METHOD INTERNAL ParseResponsePayload : DINT
VAR_INPUT
  /// Response data
  ResponseData : RobotLibraryRecvDataFB;
  /// Timestamp
  Timestamp    : SystemTime;  
END_VAR
// Table 6-566: Received CMD payload (RC to PLC) of "MeasuringInput"
// --------------------------
// Header
// --------------------------
// Byte 000 : USINT - ParSeq | State     
// Byte 001 : SINT  - AlarmMessageSeverity    
// Byte 002 : UINT  - AlarmMessageCode HB
// Byte 003 :       - AlarmMessageCode LB
// --------------------------
// Datablock
// --------------------------
// Byte 004 : BOOL      - Enabled
// Byte 005 : UINT      - MeasuringID LW LB 
// Byte 006 : USINT     - ToolNo_1
// Byte 007 : USINT     - FrameNo_1
// Byte 008 : USINT     - ToolNo_2
// Byte 009 : USINT     - FrameNo_2
// Byte 010 : REAL      - MeasuredCartesianPosition_1.X HW HB
// Byte 011 :           - MeasuredCartesianPosition_1.X HW LB
// Byte 012 :           - MeasuredCartesianPosition_1.X LW HB
// Byte 013 :           - MeasuredCartesianPosition_1.X LW LB
// Byte 014 : REAL      - MeasuredCartesianPosition_1.Y HW HB
// Byte 015 :           - MeasuredCartesianPosition_1.Y HW LB
// Byte 016 :           - MeasuredCartesianPosition_1.Y LW HB
// Byte 017 :           - MeasuredCartesianPosition_1.Y LW LB
// Byte 018 : REAL      - MeasuredCartesianPosition_1.Z HW HB
// Byte 019 :           - MeasuredCartesianPosition_1.Z HW LB
// Byte 020 :           - MeasuredCartesianPosition_1.Z LW HB
// Byte 021 :           - MeasuredCartesianPosition_1.Z LW LB
// Byte 022 : REAL      - MeasuredCartesianPosition_1.Rx HW HB
// Byte 023 :           - MeasuredCartesianPosition_1.Rx HW LB
// Byte 024 :           - MeasuredCartesianPosition_1.Rx LW HB
// Byte 025 :           - MeasuredCartesianPosition_1.Rx LW LB
// Byte 026 : REAL      - MeasuredCartesianPosition_1.Ry HW HB
// Byte 027 :           - MeasuredCartesianPosition_1.Ry HW LB
// Byte 028 :           - MeasuredCartesianPosition_1.Ry LW HB
// Byte 029 :           - MeasuredCartesianPosition_1.Ry LW LB
// Byte 030 : REAL      - MeasuredCartesianPosition_1.Rz HW HB
// Byte 031 :           - MeasuredCartesianPosition_1.Rz HW LB
// Byte 032 :           - MeasuredCartesianPosition_1.Rz LW HB
// Byte 033 :           - MeasuredCartesianPosition_1.Rz LW LB
// Byte 034 : Config    - MeasuredCartesianPosition_1.ArmConfig
// Byte 035 :           - MeasuredCartesianPosition_1.Reserve
// Byte 036 : TurnNumber- MeasuredCartesianPosition_1.TurnNumber.J1 + J2  HW HB
// Byte 037 :           - MeasuredCartesianPosition_1.TurnNumber.J3 + J4  HW LB
// Byte 038 :           - MeasuredCartesianPosition_1.TurnNumber.J5 + J6  LW LB
// Byte 039 :           - MeasuredCartesianPosition_1.TurnNumber.E1       LW LB
// Byte 040 : REAL      - MeasuredCartesianPosition_1.E1 HW HB
// Byte 041 :           - MeasuredCartesianPosition_1.E1 HW LB
// Byte 042 :           - MeasuredCartesianPosition_1.E1 LW HB
// Byte 043 :           - MeasuredCartesianPosition_1.E1 LW LB
// Byte 044 : REAL      - MeasuredJointPosition_1.J1 HW HB
// Byte 045 :           - MeasuredJointPosition_1.J1 HW LB
// Byte 046 :           - MeasuredJointPosition_1.J1 LW HB
// Byte 047 :           - MeasuredJointPosition_1.J1 LW LB
// Byte 048 : REAL      - MeasuredJointPosition_1.J2 HW HB
// Byte 049 :           - MeasuredJointPosition_1.J2 HW LB
// Byte 050 :           - MeasuredJointPosition_1.J2 LW HB
// Byte 051 :           - MeasuredJointPosition_1.J2 LW LB
// Byte 052 : REAL      - MeasuredJointPosition_1.J3 HW HB
// Byte 053 :           - MeasuredJointPosition_1.J3 HW LB
// Byte 054 :           - MeasuredJointPosition_1.J3 LW HB
// Byte 055 :           - MeasuredJointPosition_1.J3 LW LB
// Byte 056 : REAL      - MeasuredJointPosition_1.J4 HW HB
// Byte 057 :           - MeasuredJointPosition_1.J4 HW LB
// Byte 058 :           - MeasuredJointPosition_1.J4 LW HB
// Byte 059 :           - MeasuredJointPosition_1.J4 LW LB
// Byte 060 : REAL      - MeasuredJointPosition_1.J5 HW HB
// Byte 061 :           - MeasuredJointPosition_1.J5 HW LB
// Byte 062 :           - MeasuredJointPosition_1.J5 LW HB
// Byte 063 :           - MeasuredJointPosition_1.J5 LW LB
// Byte 064 : REAL      - MeasuredJointPosition_1.J6 HW HB
// Byte 065 :           - MeasuredJointPosition_1.J6 HW LB
// Byte 066 :           - MeasuredJointPosition_1.J6 LW HB
// Byte 067 :           - MeasuredJointPosition_1.J6 LW LB
// Byte 068 : REAL      - MeasuredJointPosition_1.E1 HW HB
// Byte 069 :           - MeasuredJointPosition_1.E1 HW LB
// Byte 070 :           - MeasuredJointPosition_1.E1 LW HB
// Byte 071 :           - MeasuredJointPosition_1.E1 LW LB
// Byte 072 : REAL      - MeasuredCartesianPosition_2.X HW HB
// Byte 073 :           - MeasuredCartesianPosition_2.X HW LB
// Byte 074 :           - MeasuredCartesianPosition_2.X LW HB
// Byte 075 :           - MeasuredCartesianPosition_2.X LW LB
// Byte 076 : REAL      - MeasuredCartesianPosition_2.Y HW HB
// Byte 077 :           - MeasuredCartesianPosition_2.Y HW LB
// Byte 078 :           - MeasuredCartesianPosition_2.Y LW HB
// Byte 079 :           - MeasuredCartesianPosition_2.Y LW LB
// Byte 080 : REAL      - MeasuredCartesianPosition_2.Z HW HB
// Byte 081 :           - MeasuredCartesianPosition_2.Z HW LB
// Byte 082 :           - MeasuredCartesianPosition_2.Z LW HB
// Byte 083 :           - MeasuredCartesianPosition_2.Z LW LB
// Byte 084 : REAL      - MeasuredCartesianPosition_2.Rx HW HB
// Byte 085 :           - MeasuredCartesianPosition_2.Rx HW LB
// Byte 086 :           - MeasuredCartesianPosition_2.Rx LW HB
// Byte 087 :           - MeasuredCartesianPosition_2.Rx LW LB
// Byte 088 : REAL      - MeasuredCartesianPosition_2.Ry HW HB
// Byte 089 :           - MeasuredCartesianPosition_2.Ry HW LB
// Byte 090 :           - MeasuredCartesianPosition_2.Ry LW HB
// Byte 091 :           - MeasuredCartesianPosition_2.Ry LW LB
// Byte 092 : REAL      - MeasuredCartesianPosition_2.Rz HW HB
// Byte 093 :           - MeasuredCartesianPosition_2.Rz HW LB
// Byte 094 :           - MeasuredCartesianPosition_2.Rz LW HB
// Byte 095 :           - MeasuredCartesianPosition_2.Rz LW LB
// Byte 096 : Config    - MeasuredCartesianPosition_2.ArmConfig
// Byte 097 :           - MeasuredCartesianPosition_2.Reserve
// Byte 098 : TurnNumber- MeasuredCartesianPosition_2.TurnNumber.J1 + J2  HW HB
// Byte 099 :           - MeasuredCartesianPosition_2.TurnNumber.J3 + J4  HW LB
// Byte 100 :           - MeasuredCartesianPosition_2.TurnNumber.J5 + J6  LW LB
// Byte 101 :           - MeasuredCartesianPosition_2.TurnNumber.E1       LW LB
// Byte 102 : REAL      - MeasuredCartesianPosition_2.E1 HW HB
// Byte 103 :           - MeasuredCartesianPosition_2.E1 HW LB
// Byte 104 :           - MeasuredCartesianPosition_2.E1 LW HB
// Byte 105 :           - MeasuredCartesianPosition_2.E1 LW LB
// Byte 106 : REAL      - MeasuredJointPosition_2.J1 HW HB
// Byte 107 :           - MeasuredJointPosition_2.J1 HW LB
// Byte 108 :           - MeasuredJointPosition_2.J1 LW HB
// Byte 109 :           - MeasuredJointPosition_2.J1 LW LB
// Byte 110 : REAL      - MeasuredJointPosition_2.J2 HW HB
// Byte 111 :           - MeasuredJointPosition_2.J2 HW LB
// Byte 112 :           - MeasuredJointPosition_2.J2 LW HB
// Byte 113 :           - MeasuredJointPosition_2.J2 LW LB
// Byte 114 : REAL      - MeasuredJointPosition_2.J3 HW HB
// Byte 115 :           - MeasuredJointPosition_2.J3 HW LB
// Byte 116 :           - MeasuredJointPosition_2.J3 LW HB
// Byte 117 :           - MeasuredJointPosition_2.J3 LW LB
// Byte 118 : REAL      - MeasuredJointPosition_2.J4 HW HB
// Byte 119 :           - MeasuredJointPosition_2.J4 HW LB
// Byte 120 :           - MeasuredJointPosition_2.J4 LW HB
// Byte 121 :           - MeasuredJointPosition_2.J4 LW LB
// Byte 122 : REAL      - MeasuredJointPosition_2.J5 HW HB
// Byte 123 :           - MeasuredJointPosition_2.J5 HW LB
// Byte 124 :           - MeasuredJointPosition_2.J5 LW HB
// Byte 125 :           - MeasuredJointPosition_2.J5 LW LB
// Byte 126 : REAL      - MeasuredJointPosition_2.J6 HW HB
// Byte 127 :           - MeasuredJointPosition_2.J6 HW LB
// Byte 128 :           - MeasuredJointPosition_2.J6 LW HB
// Byte 129 :           - MeasuredJointPosition_2.J6 LW LB
// Byte 130 : REAL      - MeasuredJointPosition_2.E1 HW HB
// Byte 131 :           - MeasuredJointPosition_2.E1 HW LB
// Byte 132 :           - MeasuredJointPosition_2.E1 LW HB
// Byte 133 :           - MeasuredJointPosition_2.E1 LW LB
// Byte 134 : REAL      - MeasuredCartesianPosition_1.E2 HW HB
// Byte 135 :           - MeasuredCartesianPosition_1.E2 HW LB
// Byte 136 :           - MeasuredCartesianPosition_1.E2 LW HB
// Byte 137 :           - MeasuredCartesianPosition_1.E2 LW LB
// Byte 138 : REAL      - MeasuredCartesianPosition_1.E3 HW HB
// Byte 139 :           - MeasuredCartesianPosition_1.E3 HW LB
// Byte 140 :           - MeasuredCartesianPosition_1.E3 LW HB
// Byte 141 :           - MeasuredCartesianPosition_1.E3 LW LB
// Byte 142 : REAL      - MeasuredCartesianPosition_1.E4 HW HB
// Byte 143 :           - MeasuredCartesianPosition_1.E4 HW LB
// Byte 144 :           - MeasuredCartesianPosition_1.E4 LW HB
// Byte 145 :           - MeasuredCartesianPosition_1.E4 LW LB
// Byte 146 : REAL      - MeasuredCartesianPosition_1.E5 HW HB
// Byte 147 :           - MeasuredCartesianPosition_1.E5 HW LB
// Byte 148 :           - MeasuredCartesianPosition_1.E5 LW HB
// Byte 149 :           - MeasuredCartesianPosition_1.E5 LW LB
// Byte 150 : REAL      - MeasuredCartesianPosition_1.E6 HW HB
// Byte 151 :           - MeasuredCartesianPosition_1.E6 HW LB
// Byte 152 :           - MeasuredCartesianPosition_1.E6 LW HB
// Byte 153 :           - MeasuredCartesianPosition_1.E6 LW LB
// Byte 154 : REAL      - MeasuredJointPosition_1.E2 HW HB
// Byte 155 :           - MeasuredJointPosition_1.E2 HW LB
// Byte 156 :           - MeasuredJointPosition_1.E2 LW HB
// Byte 157 :           - MeasuredJointPosition_1.E2 LW LB
// Byte 158 : REAL      - MeasuredJointPosition_1.E3 HW HB
// Byte 159 :           - MeasuredJointPosition_1.E3 HW LB
// Byte 160 :           - MeasuredJointPosition_1.E3 LW HB
// Byte 161 :           - MeasuredJointPosition_1.E3 LW LB
// Byte 162 : REAL      - MeasuredJointPosition_1.E4 HW HB
// Byte 163 :           - MeasuredJointPosition_1.E4 HW LB
// Byte 164 :           - MeasuredJointPosition_1.E4 LW HB
// Byte 165 :           - MeasuredJointPosition_1.E4 LW LB
// Byte 166 : REAL      - MeasuredJointPosition_1.E5 HW HB
// Byte 167 :           - MeasuredJointPosition_1.E5 HW LB
// Byte 168 :           - MeasuredJointPosition_1.E5 LW HB
// Byte 169 :           - MeasuredJointPosition_1.E5 LW LB
// Byte 170 : REAL      - MeasuredJointPosition_1.E6 HW HB
// Byte 171 :           - MeasuredJointPosition_1.E6 HW LB
// Byte 172 :           - MeasuredJointPosition_1.E6 LW HB
// Byte 173 :           - MeasuredJointPosition_1.E6 LW LB
// Byte 174 : REAL      - MeasuredCartesianPosition_2.E2 HW HB
// Byte 175 :           - MeasuredCartesianPosition_2.E2 HW LB
// Byte 176 :           - MeasuredCartesianPosition_2.E2 LW HB
// Byte 177 :           - MeasuredCartesianPosition_2.E2 LW LB
// Byte 178 : REAL      - MeasuredCartesianPosition_2.E3 HW HB
// Byte 179 :           - MeasuredCartesianPosition_2.E3 HW LB
// Byte 180 :           - MeasuredCartesianPosition_2.E3 LW HB
// Byte 181 :           - MeasuredCartesianPosition_2.E3 LW LB
// Byte 182 : REAL      - MeasuredCartesianPosition_2.E4 HW HB
// Byte 183 :           - MeasuredCartesianPosition_2.E4 HW LB
// Byte 184 :           - MeasuredCartesianPosition_2.E4 LW HB
// Byte 185 :           - MeasuredCartesianPosition_2.E4 LW LB
// Byte 186 : REAL      - MeasuredCartesianPosition_2.E5 HW HB
// Byte 187 :           - MeasuredCartesianPosition_2.E5 HW LB
// Byte 188 :           - MeasuredCartesianPosition_2.E5 LW HB
// Byte 189 :           - MeasuredCartesianPosition_2.E5 LW LB
// Byte 190 : REAL      - MeasuredCartesianPosition_2.E6 HW HB
// Byte 191 :           - MeasuredCartesianPosition_2.E6 HW LB
// Byte 192 :           - MeasuredCartesianPosition_2.E6 LW HB
// Byte 193 :           - MeasuredCartesianPosition_2.E6 LW LB
// Byte 194 : REAL      - MeasuredJointPosition_2.E2 HW HB
// Byte 195 :           - MeasuredJointPosition_2.E2 HW LB
// Byte 196 :           - MeasuredJointPosition_2.E2 LW HB
// Byte 197 :           - MeasuredJointPosition_2.E2 LW LB
// Byte 198 : REAL      - MeasuredJointPosition_2.E3 HW HB
// Byte 199 :           - MeasuredJointPosition_2.E3 HW LB
// Byte 200 :           - MeasuredJointPosition_2.E3 LW HB
// Byte 201 :           - MeasuredJointPosition_2.E3 LW LB
// Byte 202 : REAL      - MeasuredJointPosition_2.E4 HW HB
// Byte 203 :           - MeasuredJointPosition_2.E4 HW LB
// Byte 204 :           - MeasuredJointPosition_2.E4 LW HB
// Byte 205 :           - MeasuredJointPosition_2.E4 LW LB
// Byte 206 : REAL      - MeasuredJointPosition_2.E5 HW HB
// Byte 207 :           - MeasuredJointPosition_2.E5 HW LB
// Byte 208 :           - MeasuredJointPosition_2.E5 LW HB
// Byte 209 :           - MeasuredJointPosition_2.E5 LW LB
// Byte 210 : REAL      - MeasuredJointPosition_2.E6 HW HB
// Byte 211 :           - MeasuredJointPosition_2.E6 HW LB
// Byte 212 :           - MeasuredJointPosition_2.E6 LW HB
// Byte 213 :           - MeasuredJointPosition_2.E6 LW LB
// call base implementation to parse the header from payload buffer
ResponseData.PayloadPtr := SUPER^.ParseResponsePayload(ResponseData := ResponseData, Timestamp := Timestamp);

// copy parsed header to response
_response.ParSeq               := _rspHeader.ParSeq;
_response.State                := _rspHeader.State;
_response.AlarmMessageSeverity := _rspHeader.AlarmMessageSeverity;
_response.AlarmMessageCode     := _rspHeader.AlarmMessageCode;


// Get Response.MeasuringID
_response.MeasuringID   := ResponseData.GetUint();
// Get Response.Measurings[1].ToolNo
_response.Measurings[1].ToolNo := ResponseData.GetUsint();
// Get Response.Measurings[1].FrameNo
_response.Measurings[1].FrameNo := ResponseData.GetUsint();
// Get Response.Measurings[2].ToolNo
_response.Measurings[2].ToolNo := ResponseData.GetUsint();
// Get Response.Measurings[2].FrameNo
_response.Measurings[2].FrameNo := ResponseData.GetUsint();
// Get Response.Measurings[1].MeasuredCartesianPosition.X
_response.Measurings[1].MeasuredCartesianPosition.X := ResponseData.GetReal();
// Get Response.Measurings[1].MeasuredCartesianPosition.Y
_response.Measurings[1].MeasuredCartesianPosition.Y := ResponseData.GetReal();
// Get Response.Measurings[1].MeasuredCartesianPosition.Z
_response.Measurings[1].MeasuredCartesianPosition.Z := ResponseData.GetReal();
// Get Response.Measurings[1].MeasuredCartesianPosition.Rx
_response.Measurings[1].MeasuredCartesianPosition.Rx := ResponseData.GetReal();
// Get Response.Measurings[1].MeasuredCartesianPosition.Ry
_response.Measurings[1].MeasuredCartesianPosition.Ry := ResponseData.GetReal();
// Get Response.Measurings[1].MeasuredCartesianPosition.Rz
_response.Measurings[1].MeasuredCartesianPosition.Rz := ResponseData.GetReal();
// Get Response.Measurings[1].MeasuredCartesianPosition.Config
_response.Measurings[1].MeasuredCartesianPosition.Config := ResponseData.GetArmConfig();
// Get Response.Measurings[1].MeasuredCartesianPosition.TurnNumber
_response.Measurings[1].MeasuredCartesianPosition.TurnNumber := ResponseData.GetTurnNumbers();
// Get Response.Measurings[1].MeasuredCartesianPosition.E1
_response.Measurings[1].MeasuredCartesianPosition.E1 := ResponseData.GetReal();
// Get Response.Measurings[1].MeasuredJointPosition.J1
_response.Measurings[1].MeasuredJointPosition.J1 := ResponseData.GetReal();
// Get Response.Measurings[1].MeasuredJointPosition.J2
_response.Measurings[1].MeasuredJointPosition.J2 := ResponseData.GetReal();
// Get Response.Measurings[1].MeasuredJointPosition.J3
_response.Measurings[1].MeasuredJointPosition.J3 := ResponseData.GetReal();
// Get Response.Measurings[1].MeasuredJointPosition.J4
_response.Measurings[1].MeasuredJointPosition.J4 := ResponseData.GetReal();
// Get Response.Measurings[1].MeasuredJointPosition.J5
_response.Measurings[1].MeasuredJointPosition.J5 := ResponseData.GetReal();
// Get Response.Measurings[1].MeasuredJointPosition.J6
_response.Measurings[1].MeasuredJointPosition.J6 := ResponseData.GetReal();
// Get Response.Measurings[1].MeasuredJointPosition.E1
_response.Measurings[1].MeasuredJointPosition.E1 := ResponseData.GetReal();
// Get Response.Measurings[2].MeasuredCartesianPosition.X
_response.Measurings[2].MeasuredCartesianPosition.X := ResponseData.GetReal();
// Get Response.Measurings[2].MeasuredCartesianPosition.Y
_response.Measurings[2].MeasuredCartesianPosition.Y := ResponseData.GetReal();
// Get Response.Measurings[2].MeasuredCartesianPosition.Z
_response.Measurings[2].MeasuredCartesianPosition.Z := ResponseData.GetReal();
// Get Response.Measurings[2].MeasuredCartesianPosition.Rx
_response.Measurings[2].MeasuredCartesianPosition.Rx := ResponseData.GetReal();
// Get Response.Measurings[2].MeasuredCartesianPosition.Ry
_response.Measurings[2].MeasuredCartesianPosition.Ry := ResponseData.GetReal();
// Get Response.Measurings[2].MeasuredCartesianPosition.Rz
_response.Measurings[2].MeasuredCartesianPosition.Rz := ResponseData.GetReal();
// Get Response.Measurings[2].MeasuredCartesianPosition.Config
_response.Measurings[2].MeasuredCartesianPosition.Config := ResponseData.GetArmConfig();
// Get Response.Measurings[2].MeasuredCartesianPosition.TurnNumber
_response.Measurings[2].MeasuredCartesianPosition.TurnNumber := ResponseData.GetTurnNumbers();
// Get Response.Measurings[2].MeasuredCartesianPosition.E1
_response.Measurings[2].MeasuredCartesianPosition.E1 := ResponseData.GetReal();
// Get Response.Measurings[2].MeasuredJointPosition.J1
_response.Measurings[2].MeasuredJointPosition.J1 := ResponseData.GetReal();
// Get Response.Measurings[2].MeasuredJointPosition.J2
_response.Measurings[2].MeasuredJointPosition.J2 := ResponseData.GetReal();
// Get Response.Measurings[2].MeasuredJointPosition.J3
_response.Measurings[2].MeasuredJointPosition.J3 := ResponseData.GetReal();
// Get Response.Measurings[2].MeasuredJointPosition.J4
_response.Measurings[2].MeasuredJointPosition.J4 := ResponseData.GetReal();
// Get Response.Measurings[2].MeasuredJointPosition.J5
_response.Measurings[2].MeasuredJointPosition.J5 := ResponseData.GetReal();
// Get Response.Measurings[2].MeasuredJointPosition.J6
_response.Measurings[2].MeasuredJointPosition.J6 := ResponseData.GetReal();
// Get Response.Measurings[2].MeasuredJointPosition.E1
_response.Measurings[2].MeasuredJointPosition.E1 := ResponseData.GetReal();
// Get Response.Measurings[1].MeasuredCartesianPosition.E2
_response.Measurings[1].MeasuredCartesianPosition.E2 := ResponseData.GetReal();
// Get Response.Measurings[1].MeasuredCartesianPosition.E3
_response.Measurings[1].MeasuredCartesianPosition.E3 := ResponseData.GetReal();
// Get Response.Measurings[1].MeasuredCartesianPosition.E4
_response.Measurings[1].MeasuredCartesianPosition.E4 := ResponseData.GetReal();
// Get Response.Measurings[1].MeasuredCartesianPosition.E5
_response.Measurings[1].MeasuredCartesianPosition.E5 := ResponseData.GetReal();
// Get Response.Measurings[1].MeasuredCartesianPosition.E6
_response.Measurings[1].MeasuredCartesianPosition.E6 := ResponseData.GetReal();
// Get Response.Measurings[1].MeasuredJointPosition.E2
_response.Measurings[1].MeasuredJointPosition.E2 := ResponseData.GetReal();
// Get Response.Measurings[1].MeasuredJointPosition.E3
_response.Measurings[1].MeasuredJointPosition.E3 := ResponseData.GetReal();
// Get Response.Measurings[1].MeasuredJointPosition.E4
_response.Measurings[1].MeasuredJointPosition.E4 := ResponseData.GetReal();
// Get Response.Measurings[1].MeasuredJointPosition.E5
_response.Measurings[1].MeasuredJointPosition.E5 := ResponseData.GetReal();
// Get Response.Measurings[1].MeasuredJointPosition.E6
_response.Measurings[1].MeasuredJointPosition.E6 := ResponseData.GetReal();
// Get Response.Measurings[2].MeasuredCartesianPosition.E2
_response.Measurings[2].MeasuredCartesianPosition.E2 := ResponseData.GetReal();
// Get Response.Measurings[2].MeasuredCartesianPosition.E3
_response.Measurings[2].MeasuredCartesianPosition.E3 := ResponseData.GetReal();
// Get Response.Measurings[2].MeasuredCartesianPosition.E4
_response.Measurings[2].MeasuredCartesianPosition.E4 := ResponseData.GetReal();
// Get Response.Measurings[2].MeasuredCartesianPosition.E5
_response.Measurings[2].MeasuredCartesianPosition.E5 := ResponseData.GetReal();
// Get Response.Measurings[2].MeasuredCartesianPosition.E6
_response.Measurings[2].MeasuredCartesianPosition.E6 := ResponseData.GetReal();
// Get Response.Measurings[2].MeasuredJointPosition.E2
_response.Measurings[2].MeasuredJointPosition.E2 := ResponseData.GetReal();
// Get Response.Measurings[2].MeasuredJointPosition.E3
_response.Measurings[2].MeasuredJointPosition.E3 := ResponseData.GetReal();
// Get Response.Measurings[2].MeasuredJointPosition.E4
_response.Measurings[2].MeasuredJointPosition.E4 := ResponseData.GetReal();
// Get Response.Measurings[2].MeasuredJointPosition.E5
_response.Measurings[2].MeasuredJointPosition.E5 := ResponseData.GetReal();
// Get Response.Measurings[2].MeasuredJointPosition.E6
_response.Measurings[2].MeasuredJointPosition.E6 := ResponseData.GetReal();

// Create logging
ParseResponsePayloadLog(ResponseData := ResponseData, Timestamp := Timestamp);
END_METHOD

METHOD INTERNAL ParseResponsePayloadLog
VAR_INPUT
  /// Response data
  ResponseData : RobotLibraryRecvDataFB;
  /// Timestamp
  Timestamp    : SystemTime;  
END_VAR
VAR
  /// internal index for loops
  _idx : DINT;
END_VAR
// Create log entry for Parameter start
CreateLogMessage      ( Timestamp   := Timestamp,
                        MessageType := MessageType.CMD,
                        Severity    := Severity.DEBUG,
                        MessageCode := 0,
                        MessageText := 'Parsed the following parameter(s) from response data:');
                        
// Create log entry for MeasuringID
CreateLogMessagePara1 ( Timestamp   := Timestamp,
                        MessageType := MessageType.CMD,
                        Severity    := Severity.DEBUG,
                        MessageCode := 0,
                        MessageText := 'Response.MeasuringID = {1}',
                        Para1       :=  UINT_TO_STRING(_response.MeasuringID));

// Create log entry for MeasuringID
CreateLogMessagePara1 ( Timestamp   := Timestamp,
                        MessageType := MessageType.CMD,
                        Severity    := Severity.DEBUG,
                        MessageCode := 0,
                        MessageText := 'Response.MeasuringID = {1}',
                        Para1       :=  UINT_TO_STRING(_response.MeasuringID));

// Create log entry for Measurings[x]
FOR _idx := 1 TO 2
DO
  // Create log entry for Measurings[x].ToolNo
  CreateLogMessagePara2 ( Timestamp   := Timestamp,
                          MessageType := MessageType.CMD,
                          Severity    := Severity.DEBUG,
                          MessageCode := 0,
                          MessageText := 'Response.Measurings[{2}].ToolNo = {1}',
                          Para1       :=  USINT_TO_STRING(_response.Measurings[_idx].ToolNo),
                          Para2       :=  DINT_TO_STRING(_idx));

  // Create log entry for Measurings[x].FrameNo
  CreateLogMessagePara2 ( Timestamp   := Timestamp,
                          MessageType := MessageType.CMD,
                          Severity    := Severity.DEBUG,
                          MessageCode := 0,
                          MessageText := 'Response.Measurings[{2}].FrameNo = {1}',
                          Para1       :=  USINT_TO_STRING(_response.Measurings[_idx].FrameNo),
                          Para2       :=  DINT_TO_STRING(_idx));
END_FOR


// Create log entry for Measurings[x]
FOR _idx := 1 TO 2
DO
  // Create log entry for Measurings[x].MeasuredCartesianPosition.X
  CreateLogMessagePara2 ( Timestamp   := Timestamp,
                          MessageType := MessageType.CMD,
                          Severity    := Severity.DEBUG,
                          MessageCode := 0,
                          MessageText := 'Response.Measurings[{2}].MeasuredCartesianPosition.X = {1}',
                          Para1       :=  REAL_TO_STRING(_response.Measurings[_idx].MeasuredCartesianPosition.X),
                          Para2       :=  DINT_TO_STRING(_idx));

  // Create log entry for Measurings[x].MeasuredCartesianPosition.Y
  CreateLogMessagePara2 ( Timestamp   := Timestamp,
                          MessageType := MessageType.CMD,
                          Severity    := Severity.DEBUG,
                          MessageCode := 0,
                          MessageText := 'Response.Measurings[{2}].MeasuredCartesianPosition.Y = {1}',
                          Para1       :=  REAL_TO_STRING(_response.Measurings[_idx].MeasuredCartesianPosition.Y),
                          Para2       :=  DINT_TO_STRING(_idx));
                          
  // Create log entry for Measurings[x].MeasuredCartesianPosition.Z
  CreateLogMessagePara2 ( Timestamp   := Timestamp,
                          MessageType := MessageType.CMD,
                          Severity    := Severity.DEBUG,
                          MessageCode := 0,
                          MessageText := 'Response.Measurings[{2}].MeasuredCartesianPosition.Z = {1}',
                          Para1       :=  REAL_TO_STRING(_response.Measurings[_idx].MeasuredCartesianPosition.Z),
                          Para2       :=  DINT_TO_STRING(_idx));
                          
  // Create log entry for Measurings[x].MeasuredCartesianPosition.Rx
  CreateLogMessagePara2 ( Timestamp   := Timestamp,
                          MessageType := MessageType.CMD,
                          Severity    := Severity.DEBUG,
                          MessageCode := 0,
                          MessageText := 'Response.Measurings[{2}].MeasuredCartesianPosition.Rx = {1}',
                          Para1       :=  REAL_TO_STRING(_response.Measurings[_idx].MeasuredCartesianPosition.Rx),
                          Para2       :=  DINT_TO_STRING(_idx));

  // Create log entry for Measurings[x].MeasuredCartesianPosition.Ry
  CreateLogMessagePara2 ( Timestamp   := Timestamp,
                          MessageType := MessageType.CMD,
                          Severity    := Severity.DEBUG,
                          MessageCode := 0,
                          MessageText := 'Response.Measurings[{2}].MeasuredCartesianPosition.Ry = {1}',
                          Para1       :=  REAL_TO_STRING(_response.Measurings[_idx].MeasuredCartesianPosition.Ry),
                          Para2       :=  DINT_TO_STRING(_idx));

  // Create log entry for Measurings[x].MeasuredCartesianPosition.Rz
  CreateLogMessagePara2 ( Timestamp   := Timestamp,
                          MessageType := MessageType.CMD,
                          Severity    := Severity.DEBUG,
                          MessageCode := 0,
                          MessageText := 'Response.Measurings[{2}].MeasuredCartesianPosition.Rz = {1}',
                          Para1       :=  REAL_TO_STRING(_response.Measurings[_idx].MeasuredCartesianPosition.Rz),
                          Para2       :=  DINT_TO_STRING(_idx));

  // Create log entry for Measurings[x].MeasuredCartesianPosition.Config
  CreateLogMessagePara2 ( Timestamp   := Timestamp,
                          MessageType := MessageType.CMD,
                          Severity    := Severity.DEBUG,
                          MessageCode := 0,
                          MessageText := 'Response.Measurings[{2}].MeasuredCartesianPosition.Config = {1}',
                          Para1       :=  ARM_CONFIG_TO_STRING(_response.Measurings[_idx].MeasuredCartesianPosition.Config),
                          Para2       :=  DINT_TO_STRING(_idx));

  // Create log entry for Measurings[x].MeasuredCartesianPosition.TurnNumber.J1Turns
  CreateLogMessagePara2 ( Timestamp   := Timestamp,
                          MessageType := MessageType.CMD,
                          Severity    := Severity.DEBUG,
                          MessageCode := 0,
                          MessageText := 'Response.Measurings[{2}].MeasuredCartesianPosition.TurnNumber.J1Turns = {1}',
                          Para1       :=  SINT_TO_STRING(_response.Measurings[_idx].MeasuredCartesianPosition.TurnNumber.J1Turns),
                          Para2       :=  DINT_TO_STRING(_idx));

  // Create log entry for Measurings[x].MeasuredCartesianPosition.TurnNumber.J2Turns
  CreateLogMessagePara2 ( Timestamp   := Timestamp,
                          MessageType := MessageType.CMD,
                          Severity    := Severity.DEBUG,
                          MessageCode := 0,
                          MessageText := 'Response.Measurings[{2}].MeasuredCartesianPosition.TurnNumber.J2Turns = {1}',
                          Para1       :=  SINT_TO_STRING(_response.Measurings[_idx].MeasuredCartesianPosition.TurnNumber.J2Turns),
                          Para2       :=  DINT_TO_STRING(_idx));

  // Create log entry for Measurings[x].MeasuredCartesianPosition.TurnNumber.J3Turns
  CreateLogMessagePara2 ( Timestamp   := Timestamp,
                          MessageType := MessageType.CMD,
                          Severity    := Severity.DEBUG,
                          MessageCode := 0,
                          MessageText := 'Response.Measurings[{2}].MeasuredCartesianPosition.TurnNumber.J3Turns = {1}',
                          Para1       :=  SINT_TO_STRING(_response.Measurings[_idx].MeasuredCartesianPosition.TurnNumber.J3Turns),
                          Para2       :=  DINT_TO_STRING(_idx));
                          
  // Create log entry for Measurings[x].MeasuredCartesianPosition.TurnNumber.J4Turns
  CreateLogMessagePara2 ( Timestamp   := Timestamp,
                          MessageType := MessageType.CMD,
                          Severity    := Severity.DEBUG,
                          MessageCode := 0,
                          MessageText := 'Response.Measurings[{2}].MeasuredCartesianPosition.TurnNumber.J4Turns = {1}',
                          Para1       :=  SINT_TO_STRING(_response.Measurings[_idx].MeasuredCartesianPosition.TurnNumber.J4Turns),
                          Para2       :=  DINT_TO_STRING(_idx));

  // Create log entry for Measurings[x].MeasuredCartesianPosition.TurnNumber.J5Turns
  CreateLogMessagePara2 ( Timestamp   := Timestamp,
                          MessageType := MessageType.CMD,
                          Severity    := Severity.DEBUG,
                          MessageCode := 0,
                          MessageText := 'Response.Measurings[{2}].MeasuredCartesianPosition.TurnNumber.J5Turns = {1}',
                          Para1       :=  SINT_TO_STRING(_response.Measurings[_idx].MeasuredCartesianPosition.TurnNumber.J5Turns),
                          Para2       :=  DINT_TO_STRING(_idx));
                          
  // Create log entry for Measurings[x].MeasuredCartesianPosition.TurnNumber.J6Turns
  CreateLogMessagePara2 ( Timestamp   := Timestamp,
                          MessageType := MessageType.CMD,
                          Severity    := Severity.DEBUG,
                          MessageCode := 0,
                          MessageText := 'Response.Measurings[{2}].MeasuredCartesianPosition.TurnNumber.J6Turns = {1}',
                          Para1       :=  SINT_TO_STRING(_response.Measurings[_idx].MeasuredCartesianPosition.TurnNumber.J6Turns),
                          Para2       :=  DINT_TO_STRING(_idx));

  // Create log entry for Measurings[x].MeasuredCartesianPosition.TurnNumber.E1Turns
  CreateLogMessagePara2 ( Timestamp   := Timestamp,
                          MessageType := MessageType.CMD,
                          Severity    := Severity.DEBUG,
                          MessageCode := 0,
                          MessageText := 'Response.Measurings[{2}].MeasuredCartesianPosition.TurnNumber.E1Turns = {1}',
                          Para1       :=  SINT_TO_STRING(_response.Measurings[_idx].MeasuredCartesianPosition.TurnNumber.E1Turns),
                          Para2       :=  DINT_TO_STRING(_idx));

  // Create log entry for Measurings[x].MeasuredCartesianPosition.E1
  CreateLogMessagePara2 ( Timestamp   := Timestamp,
                          MessageType := MessageType.CMD,
                          Severity    := Severity.DEBUG,
                          MessageCode := 0,
                          MessageText := 'Response.Measurings[{2}].MeasuredCartesianPosition.E1 = {1}',
                          Para1       :=  REAL_TO_STRING(_response.Measurings[_idx].MeasuredCartesianPosition.E1),
                          Para2       :=  DINT_TO_STRING(_idx));
                          
  // Create log entry for Measurings[x].MeasuredJointPosition.J1
  CreateLogMessagePara2 ( Timestamp   := Timestamp,
                          MessageType := MessageType.CMD,
                          Severity    := Severity.DEBUG,
                          MessageCode := 0,
                          MessageText := 'Response.Measurings[{2}].MeasuredJointPosition.J1 = {1}',
                          Para1       :=  REAL_TO_STRING(_response.Measurings[_idx].MeasuredJointPosition.J1),
                          Para2       :=  DINT_TO_STRING(_idx));
                          
  // Create log entry for Measurings[x].MeasuredJointPosition.J2
  CreateLogMessagePara2 ( Timestamp   := Timestamp,
                          MessageType := MessageType.CMD,
                          Severity    := Severity.DEBUG,
                          MessageCode := 0,
                          MessageText := 'Response.Measurings[{2}].MeasuredJointPosition.J2 = {1}',
                          Para1       :=  REAL_TO_STRING(_response.Measurings[_idx].MeasuredJointPosition.J2),
                          Para2       :=  DINT_TO_STRING(_idx));

  // Create log entry for Measurings[x].MeasuredJointPosition.J3
  CreateLogMessagePara2 ( Timestamp   := Timestamp,
                          MessageType := MessageType.CMD,
                          Severity    := Severity.DEBUG,
                          MessageCode := 0,
                          MessageText := 'Response.Measurings[{2}].MeasuredJointPosition.J3 = {1}',
                          Para1       :=  REAL_TO_STRING(_response.Measurings[_idx].MeasuredJointPosition.J3),
                          Para2       :=  DINT_TO_STRING(_idx));
                          
  // Create log entry for Measurings[x].MeasuredJointPosition.J4
  CreateLogMessagePara2 ( Timestamp   := Timestamp,
                          MessageType := MessageType.CMD,
                          Severity    := Severity.DEBUG,
                          MessageCode := 0,
                          MessageText := 'Response.Measurings[{2}].MeasuredJointPosition.J4 = {1}',
                          Para1       :=  REAL_TO_STRING(_response.Measurings[_idx].MeasuredJointPosition.J4),
                          Para2       :=  DINT_TO_STRING(_idx));

  // Create log entry for Measurings[x].MeasuredJointPosition.J5
  CreateLogMessagePara2 ( Timestamp   := Timestamp,
                          MessageType := MessageType.CMD,
                          Severity    := Severity.DEBUG,
                          MessageCode := 0,
                          MessageText := 'Response.Measurings[{2}].MeasuredJointPosition.J5 = {1}',
                          Para1       :=  REAL_TO_STRING(_response.Measurings[_idx].MeasuredJointPosition.J5),
                          Para2       :=  DINT_TO_STRING(_idx));
                          
  // Create log entry for Measurings[x].MeasuredJointPosition.J6
  CreateLogMessagePara2 ( Timestamp   := Timestamp,
                          MessageType := MessageType.CMD,
                          Severity    := Severity.DEBUG,
                          MessageCode := 0,
                          MessageText := 'Response.Measurings[{2}].MeasuredJointPosition.J6 = {1}',
                          Para1       :=  REAL_TO_STRING(_response.Measurings[_idx].MeasuredJointPosition.J6),
                          Para2       :=  DINT_TO_STRING(_idx));

  // Create log entry for Measurings[x].MeasuredJointPosition.E1
  CreateLogMessagePara2 ( Timestamp   := Timestamp,
                          MessageType := MessageType.CMD,
                          Severity    := Severity.DEBUG,
                          MessageCode := 0,
                          MessageText := 'Response.Measurings[{2}].MeasuredJointPosition.E1 = {1}',
                          Para1       :=  REAL_TO_STRING(_response.Measurings[_idx].MeasuredJointPosition.E1),
                          Para2       :=  DINT_TO_STRING(_idx));
END_FOR


// Create log entry for Measurings[x]
FOR _idx := 1 TO 2
DO
  // Create log entry for Measurings[x].MeasuredCartesianPosition.E2
  CreateLogMessagePara2 ( Timestamp   := Timestamp,
                          MessageType := MessageType.CMD,
                          Severity    := Severity.DEBUG,
                          MessageCode := 0,
                          MessageText := 'Response.Measurings[{2}].MeasuredCartesianPosition.E2 = {1}',
                          Para1       :=  REAL_TO_STRING(_response.Measurings[_idx].MeasuredCartesianPosition.E2),
                          Para2       :=  DINT_TO_STRING(_idx));

  // Create log entry for Measurings[x].MeasuredCartesianPosition.E3
  CreateLogMessagePara2 ( Timestamp   := Timestamp,
                          MessageType := MessageType.CMD,
                          Severity    := Severity.DEBUG,
                          MessageCode := 0,
                          MessageText := 'Response.Measurings[{2}].MeasuredCartesianPosition.E3 = {1}',
                          Para1       :=  REAL_TO_STRING(_response.Measurings[_idx].MeasuredCartesianPosition.E3),
                          Para2       :=  DINT_TO_STRING(_idx));
                          
  // Create log entry for Measurings[x].MeasuredCartesianPosition.E4
  CreateLogMessagePara2 ( Timestamp   := Timestamp,
                          MessageType := MessageType.CMD,
                          Severity    := Severity.DEBUG,
                          MessageCode := 0,
                          MessageText := 'Response.Measurings[{2}].MeasuredCartesianPosition.E4 = {1}',
                          Para1       :=  REAL_TO_STRING(_response.Measurings[_idx].MeasuredCartesianPosition.E4),
                          Para2       :=  DINT_TO_STRING(_idx));
                          
  // Create log entry for Measurings[x].MeasuredCartesianPosition.E5
  CreateLogMessagePara2 ( Timestamp   := Timestamp,
                          MessageType := MessageType.CMD,
                          Severity    := Severity.DEBUG,
                          MessageCode := 0,
                          MessageText := 'Response.Measurings[{2}].MeasuredCartesianPosition.E5 = {1}',
                          Para1       :=  REAL_TO_STRING(_response.Measurings[_idx].MeasuredCartesianPosition.E5),
                          Para2       :=  DINT_TO_STRING(_idx));
                          
  // Create log entry for Measurings[x].MeasuredCartesianPosition.E6
  CreateLogMessagePara2 ( Timestamp   := Timestamp,
                          MessageType := MessageType.CMD,
                          Severity    := Severity.DEBUG,
                          MessageCode := 0,
                          MessageText := 'Response.Measurings[{2}].MeasuredCartesianPosition.E6 = {1}',
                          Para1       :=  REAL_TO_STRING(_response.Measurings[_idx].MeasuredCartesianPosition.E6),
                          Para2       :=  DINT_TO_STRING(_idx));

  // Create log entry for Measurings[x].MeasuredJointPosition.E2
  CreateLogMessagePara2 ( Timestamp   := Timestamp,
                          MessageType := MessageType.CMD,
                          Severity    := Severity.DEBUG,
                          MessageCode := 0,
                          MessageText := 'Response.Measurings[{2}].MeasuredJointPosition.E2 = {1}',
                          Para1       :=  REAL_TO_STRING(_response.Measurings[_idx].MeasuredJointPosition.E2),
                          Para2       :=  DINT_TO_STRING(_idx));

  // Create log entry for Measurings[x].MeasuredJointPosition.E3
  CreateLogMessagePara2 ( Timestamp   := Timestamp,
                          MessageType := MessageType.CMD,
                          Severity    := Severity.DEBUG,
                          MessageCode := 0,
                          MessageText := 'Response.Measurings[{2}].MeasuredJointPosition.E3 = {1}',
                          Para1       :=  REAL_TO_STRING(_response.Measurings[_idx].MeasuredJointPosition.E3),
                          Para2       :=  DINT_TO_STRING(_idx));
                          
  // Create log entry for Measurings[x].MeasuredJointPosition.E4
  CreateLogMessagePara2 ( Timestamp   := Timestamp,
                          MessageType := MessageType.CMD,
                          Severity    := Severity.DEBUG,
                          MessageCode := 0,
                          MessageText := 'Response.Measurings[{2}].MeasuredJointPosition.E4 = {1}',
                          Para1       :=  REAL_TO_STRING(_response.Measurings[_idx].MeasuredJointPosition.E4),
                          Para2       :=  DINT_TO_STRING(_idx));
                          
  // Create log entry for Measurings[x].MeasuredJointPosition.E5
  CreateLogMessagePara2 ( Timestamp   := Timestamp,
                          MessageType := MessageType.CMD,
                          Severity    := Severity.DEBUG,
                          MessageCode := 0,
                          MessageText := 'Response.Measurings[{2}].MeasuredJointPosition.E5 = {1}',
                          Para1       :=  REAL_TO_STRING(_response.Measurings[_idx].MeasuredJointPosition.E5),
                          Para2       :=  DINT_TO_STRING(_idx));
                          
  // Create log entry for Measurings[x].MeasuredJointPosition.E6
  CreateLogMessagePara2 ( Timestamp   := Timestamp,
                          MessageType := MessageType.CMD,
                          Severity    := Severity.DEBUG,
                          MessageCode := 0,
                          MessageText := 'Response.Measurings[{2}].MeasuredJointPosition.E6 = {1}',
                          Para1       :=  REAL_TO_STRING(_response.Measurings[_idx].MeasuredJointPosition.E6),
                          Para2       :=  DINT_TO_STRING(_idx));
                     
END_FOR
END_METHOD

METHOD PROTECTED Reset : DINT
VAR_INPUT
END_VAR
Reset := SUPER^.Reset();

Done               := FALSE;
Busy               := FALSE;
CommandBuffered    := FALSE;
END_METHOD

END_FUNCTION_BLOCK

// Library/POUs/Additional/MC_OpenBrake/MC_OpenBrakeFB
/// Release robot arm’s brakes.
FUNCTION_BLOCK MC_OpenBrakeFB EXTENDS RobotLibraryBaseExecuteFB
// ------------------------------------------------------------------------- 
//  SRCI Robot Library                                                
// ------------------------------------------------------------------------- 
//                                                                           
//  Object:      OpenBrakeFB                                       
//  Author:      Thorsten Brach                                                
//  Date:        2024-06-01
//
//  Description:                                              
//   
//                                                                           
//  Copyright: 
//    (C) 2024 Thorsten Brach. All rights reserved                                                                                                                                            
//             Licensed under the LGPL-3.0 license.
//                                                                           
//  Disclaimer:                                                                           
//    This project is provided without any guarantee and can be used for   
//    private and commercial purposes. Any use is at the user’s 
//    own risk and responsibility.
//
// -------------------------------------------------------------------------
VAR_INPUT
  /// Command parameter 
  ParCmd             : OpenBrakeParCmd;  
END_VAR

VAR_OUTPUT
  /// Command is transferred and confirmed by the RC
  CommandBuffered   : BOOL;
  /// Receiving of input parameter values has been acknowledged by RC
  ParameterAccepted : BOOL;
  /// Command output 
  OutCmd            : OpenBrakeOutCmd;  
END_VAR

VAR
  /// internal copy of command parameter 
 _parCmd             : OpenBrakeParCmd;
  /// command data to send
 _command            : OpenBrakeSendData;
  /// response data received
 _response           : OpenBrakeRecvData;      
END_VAR

SUPER^(AxesGroup := AxesGroup);

METHOD PROTECTED CheckFunctionSupported : BOOL
VAR_IN_OUT
  /// Robot assignment of function
  AxesGroup : AxesGroup; 
END_VAR
CheckFunctionSupported := AxesGroup.InternalData.RCSupportedFunctions.OpenBrake;

IF ( NOT CheckFunctionSupported )
THEN
  // call base implementation for set error and create log entry
  SUPER^.CheckFunctionSupported(AxesGroup := AxesGroup);
END_IF
END_METHOD

METHOD PROTECTED CheckParameterChanged : BOOL
VAR_IN_OUT
  /// Robot assignment of function
  AxesGroup    : AxesGroup; 
END_VAR
// Check ParCmd Size is > 0, because MemCmp does not work correctly with size = 0
IF (SIZEOF(ParCmd) = 0) 
THEN 
  RETURN;
END_IF

// compare memory 
_parameterChanged := ( SysDepMemCmp(pData1 := ADR(ParCmd), pData2 := ADR(_parCmd), DataLen := SIZEOF(ParCmd)) <> RobotLibraryConstants.OK );

// check parameter valid ?
_parameterValid   := CheckParameterValid( AxesGroup := AxesGroup );

IF ((  _parameterChanged        )  AND 
    (  _parameterValid          )) OR
    (  _parameterUpdateInternal )  
THEN  
  // reset internal flag for send parameter update
 _parameterUpdateInternal := FALSE;
  // update internal copy of parameters 
 _parCmd := ParCmd;
  // inc parameter sequence
 _command.ParSeq := _command.ParSeq + 1;
  // update command data  
  CommandData := CreateCommandPayload(AxesGroup := AxesGroup); // ( Access via reference to rCommandFB in ACR )
  // notify active command register 
  AxesGroup.Acyclic.ActiveCommandRegister.NotifyParameterChanged := _uniqueID;
  // Reset parameter accepted flag
  ParameterAccepted := FALSE;
END_IF
END_METHOD

METHOD INTERNAL CreateCommandPayload : RobotLibrarySendDataFB
VAR_IN_OUT
  /// Robot assignment of function
  AxesGroup : AxesGroup; 
END_VAR
// Table 6-681: Sent CMD payload (PLC to RC) of "OpenBrake"
// --------------------------
// Header
// --------------------------
// Byte 00 : UINT  - Type HB     
// Byte 01 :       - Type LB    
// Byte 02 : USINT - Reserve | ExecutionMode
// Byte 03 : USINT - ParSeq  | Priority
// --------------------------
// Datablock
// --------------------------
// Byte 04 : BYTE  - RobotAxesBrakeRelease
// Byte 05 : BYTE  - ExternalAxesBrakeRelease
// --------------------------
// set command parameter 
_command.CmdTyp                     :=  CmdType.OpenBrake;
_command.ExecMode                   :=  ExecMode;
_command.ParSeq                     := _command.ParSeq;
_command.Priority                   :=  Priority;
_command.RobotAxesBrakeRelease.0    := _parCmd.RobotAxesBrakeRelease   .Bit00;
_command.RobotAxesBrakeRelease.1    := _parCmd.RobotAxesBrakeRelease   .AxisJ1;
_command.RobotAxesBrakeRelease.2    := _parCmd.RobotAxesBrakeRelease   .AxisJ2;
_command.RobotAxesBrakeRelease.3    := _parCmd.RobotAxesBrakeRelease   .AxisJ3;
_command.RobotAxesBrakeRelease.4    := _parCmd.RobotAxesBrakeRelease   .AxisJ4;
_command.RobotAxesBrakeRelease.5    := _parCmd.RobotAxesBrakeRelease   .AxisJ5;
_command.RobotAxesBrakeRelease.6    := _parCmd.RobotAxesBrakeRelease   .AxisJ6;
_command.RobotAxesBrakeRelease.7    := _parCmd.RobotAxesBrakeRelease   .Bit07;
_command.ExternalAxesBrakeRelease.0 := _parCmd.ExternalAxesBrakeRelease.Bit00;
_command.ExternalAxesBrakeRelease.1 := _parCmd.ExternalAxesBrakeRelease.AxisE1;
_command.ExternalAxesBrakeRelease.2 := _parCmd.ExternalAxesBrakeRelease.AxisE2;
_command.ExternalAxesBrakeRelease.3 := _parCmd.ExternalAxesBrakeRelease.AxisE3;
_command.ExternalAxesBrakeRelease.4 := _parCmd.ExternalAxesBrakeRelease.AxisE4;
_command.ExternalAxesBrakeRelease.5 := _parCmd.ExternalAxesBrakeRelease.AxisE5;
_command.ExternalAxesBrakeRelease.6 := _parCmd.ExternalAxesBrakeRelease.AxisE6;
_command.ExternalAxesBrakeRelease.7 := _parCmd.ExternalAxesBrakeRelease.Bit07;


// copy command data to header
_cmdHeader := _command;
// call base implementation to copy header to payload buffer
CreateCommandPayload := SUPER^.CreateCommandPayload(AxesGroup := AxesGroup);

// add command.EmitterID[0]
CreateCommandPayload.AddByte(_command.RobotAxesBrakeRelease);
// add command.EmitterID[1]
CreateCommandPayload.AddByte(_command.ExternalAxesBrakeRelease);

// Create logging
CreateCommandPayloadLog(AxesGroup := AxesGroup);
END_METHOD

METHOD INTERNAL CreateCommandPayloadLog
VAR_IN_OUT
  /// Robot assignment of function
  AxesGroup : AxesGroup; 
END_VAR
// Create log entry for Parameter start
CreateLogMessage      ( Timestamp   := AxesGroup.InternalData.SystemTime,
                        MessageType := MessageType.CMD,
                        Severity    := Severity.DEBUG,
                        MessageCode := 0,
                        MessageText := 'Create command payload with the following parameter(s) :');
  
// Create log entry for RobotAxesBrakeRelease
CreateLogMessagePara1 ( Timestamp   := AxesGroup.InternalData.SystemTime,
                        MessageType := MessageType.CMD,
                        Severity    := Severity.DEBUG,
                        MessageCode := 0,
                        MessageText := 'Command.RobotAxesBrakeRelease = {1}',
                        Para1       :=  BYTE_TO_STRING_BIN(_command.RobotAxesBrakeRelease));
                        
// Create log entry for ExternalAxesBrakeRelease
CreateLogMessagePara1 ( Timestamp   := AxesGroup.InternalData.SystemTime,
                        MessageType := MessageType.CMD,
                        Severity    := Severity.DEBUG,
                        MessageCode := 0,
                        MessageText := 'Command.ExternalAxesBrakeRelease = {1}',
                        Para1       :=  BYTE_TO_STRING_BIN(_command.ExternalAxesBrakeRelease));
END_METHOD

METHOD FB_init : BOOL
VAR_INPUT
  /// if TRUE, the retain variables are initialized (warm start / cold start)
  bInitRetains : BOOL; 
  /// if TRUE, the instance afterwards gets moved into the copy code (online change)
  bInCopyCode  : BOOL;  
END_VAR
MyType := 'MC_OpenBrakeFB';

ExecMode := ExecutionMode.PARALLEL;
END_METHOD

METHOD PROTECTED OnCall
VAR_IN_OUT
  /// Robot assignment of function
  AxesGroup : AxesGroup; 
END_VAR
// call base implementation
SUPER^.OnCall(AxesGroup := AxesGroup);

CASE _stepCmd OF
  
  00:  IF ( _execute_R.Q )  
       THEN
         // Check function is supported and parameter are valid ?
         IF (( CheckFunctionSupported( AxesGroup := AxesGroup )) AND
             ( CheckParameterValid   ( AxesGroup := AxesGroup )))      
         THEN
           // set busy flag
           Busy := TRUE;
           // Reset command outputs
           SysDepMemSet(pDest := ADR(OutCmd), Value := 0, DataLen := SIZEOF(OutCmd));         
           // apply command parameter
          _parCmd := ParCmd;
           // init parameter sequence
          _command.ParSeq := 1;
           // create command data
           CommandData := CreateCommandPayload(AxesGroup := AxesGroup);
           // Add command to active command register
          _uniqueID := AxesGroup.Acyclic.ActiveCommandRegister.AddCmd( pCommandFB := ADR(THIS^ ));     
           // set timeout
           SetTimeout(PT := _timeoutCmd, rTimer := _timerCmd);
           // inc step counter
          _stepCmd := _stepCmd + 1;
         END_IF 
       END_IF
     

  01:  // Wait for responce received
       IF ( _responseReceived )
       THEN
         // reset response received flag
        _responseReceived := FALSE;

         CASE  _response.State 
         OF
           CmdMessageState.BUFFERED    : CommandBuffered    := TRUE;
           CmdMessageState.ACTIVE      : ParameterAccepted  := TRUE;           
           CmdMessageState.DONE        : Done               := TRUE;           
           CmdMessageState.ERROR       : Error              := TRUE;
         END_CASE

                
         // Done, Aborted or Error ?
         IF (_response.State >= CmdMessageState.DONE )
         THEN
           // Reset Busy flag
           Busy := FALSE;
           // Update results
           OutCmd.Enabled                          := _response.Enabled.0;
           OutCmd.RobotAxesBrakeReleased.Bit00     := _response.RobotAxesBrakeReleased.0;
           OutCmd.RobotAxesBrakeReleased.AxisJ1    := _response.RobotAxesBrakeReleased.1;
           OutCmd.RobotAxesBrakeReleased.AxisJ2    := _response.RobotAxesBrakeReleased.2;
           OutCmd.RobotAxesBrakeReleased.AxisJ3    := _response.RobotAxesBrakeReleased.3;
           OutCmd.RobotAxesBrakeReleased.AxisJ4    := _response.RobotAxesBrakeReleased.4;
           OutCmd.RobotAxesBrakeReleased.AxisJ5    := _response.RobotAxesBrakeReleased.5;
           OutCmd.RobotAxesBrakeReleased.AxisJ6    := _response.RobotAxesBrakeReleased.6;
           OutCmd.RobotAxesBrakeReleased.Bit07     := _response.RobotAxesBrakeReleased.7;
           OutCmd.ExternalAxesBrakeReleased.Bit00  := _response.ExternalAxesBrakeReleased.0;
           OutCmd.ExternalAxesBrakeReleased.AxisE1 := _response.ExternalAxesBrakeReleased.1;
           OutCmd.ExternalAxesBrakeReleased.AxisE2 := _response.ExternalAxesBrakeReleased.2;
           OutCmd.ExternalAxesBrakeReleased.AxisE3 := _response.ExternalAxesBrakeReleased.3;
           OutCmd.ExternalAxesBrakeReleased.AxisE4 := _response.ExternalAxesBrakeReleased.4;
           OutCmd.ExternalAxesBrakeReleased.AxisE5 := _response.ExternalAxesBrakeReleased.5;
           OutCmd.ExternalAxesBrakeReleased.AxisE6 := _response.ExternalAxesBrakeReleased.6;
           OutCmd.ExternalAxesBrakeReleased.Bit07  := _response.ExternalAxesBrakeReleased.7;

           // set timeout
           SetTimeout(PT := _timeoutCmd, rTimer := _timerCmd);
           // inc step counter
          _stepCmd := _stepCmd + 1; 
         END_IF
       END_IF

  02: IF ( NOT Execute)
      THEN
        Reset();
      END_IF     
ELSE
  // invalid step
  ErrorID := RobotLibraryEvents.ERR_INVALID_STEP;
END_CASE



// Reset FB
IF ( NOT Execute )
THEN
  Reset();  
END_IF
END_METHOD

METHOD INTERNAL ParseResponsePayload : DINT
VAR_INPUT
  /// Response data
  ResponseData : RobotLibraryRecvDataFB;
  /// Timestamp
  Timestamp    : SystemTime;  
END_VAR
// Table 6-682: Received CMD payload (RC to PLC) of "OpenBrake"
// --------------------------
// Header
// --------------------------
// Byte 00 : USINT - ParSeq | State     
// Byte 01 : SINT  - AlarmMessageSeverity    
// Byte 02 : UINT  - AlarmMessageCode HB
// Byte 03 :       - AlarmMessageCode LB
// --------------------------
// Datablock
// --------------------------
// Byte 04 : BOOL  - Enabled
// Byte 05 : BYTE  - RobotAxesBrakeReleased
// Byte 06 : BYTE  - ExternalAxesBrakeReleased
// --------------------------
// call base implementation to parse the header from payload buffer
ResponseData.PayloadPtr := SUPER^.ParseResponsePayload(ResponseData := ResponseData, Timestamp := Timestamp);

// copy parsed header to response
_response.ParSeq               := _rspHeader.ParSeq;
_response.State                := _rspHeader.State;
_response.AlarmMessageSeverity := _rspHeader.AlarmMessageSeverity;
_response.AlarmMessageCode     := _rspHeader.AlarmMessageCode;

// Get RobotAxesStatus
_response.RobotAxesBrakeReleased     := ResponseData.GetByte();
// Get ExternalAxesStatus
_response.ExternalAxesBrakeReleased  := ResponseData.GetByte();

// Create logging
ParseResponsePayloadLog(ResponseData := ResponseData, Timestamp := Timestamp);
END_METHOD

METHOD INTERNAL ParseResponsePayloadLog
VAR_INPUT
  /// Response data
  ResponseData : RobotLibraryRecvDataFB;
  /// Timestamp
  Timestamp    : SystemTime;  
END_VAR
// Create log entry for Parameter start
CreateLogMessage      ( Timestamp   := Timestamp,
                        MessageType := MessageType.CMD,
                        Severity    := Severity.DEBUG,
                        MessageCode := 0,
                        MessageText := 'Parsed the following parameter(s) from response data:');
                        

// Create log entry for RobotAxesBrakeReleased
CreateLogMessagePara1 ( Timestamp   := Timestamp,
                        MessageType := MessageType.CMD,
                        Severity    := Severity.DEBUG,
                        MessageCode := 0,
                        MessageText := 'Response.RobotAxesBrakeReleased = {1}',
                        Para1       :=  BYTE_TO_STRING_BIN(_response.RobotAxesBrakeReleased));

// Create log entry for ExternalAxesBrakeReleased
CreateLogMessagePara1 ( Timestamp   := Timestamp,
                        MessageType := MessageType.CMD,
                        Severity    := Severity.DEBUG,
                        MessageCode := 0,
                        MessageText := 'Response.ExternalAxesBrakeReleased = {1}',
                        Para1       :=  BYTE_TO_STRING_BIN(_response.ExternalAxesBrakeReleased));
END_METHOD

METHOD PROTECTED Reset : DINT
VAR_INPUT
END_VAR
Reset := SUPER^.Reset();

Done               := FALSE;
Busy               := FALSE;
CommandBuffered    := FALSE;
ParameterAccepted  := FALSE;
END_METHOD

END_FUNCTION_BLOCK

// Library/POUs/Additional/MC_PathAccuracyMode/MC_PathAccuracyModeFB
/// Switch path mode between high and low accuracy
FUNCTION_BLOCK MC_PathAccuracyModeFB EXTENDS RobotLibraryBaseEnableFB
// ------------------------------------------------------------------------- 
//  SRCI Robot Library                                                
// ------------------------------------------------------------------------- 
//                                                                           
//  Object:      PathAccuracyModeFB                                       
//  Author:      Thorsten Brach                                                
//  Date:        2024-06-01
//
//  Description:                                              
//   
//                                                                           
//  Copyright: 
//    (C) 2024 Thorsten Brach. All rights reserved                                                                                                                                            
//             Licensed under the LGPL-3.0 license.
//                                                                           
//  Disclaimer:                                                                           
//    This project is provided without any guarantee and can be used for   
//    private and commercial purposes. Any use is at the user’s 
//    own risk and responsibility.
//
// -------------------------------------------------------------------------
VAR_INPUT
  /// Command parameter 
  ParCmd            : PathAccuracyModeParCmd;
END_VAR

VAR_OUTPUT
  /// Command is transferred and confirmed by the RC
  CommandBuffered   : BOOL;
  /// Receiving of input parameter values has been acknowledged by RC
  ParameterAccepted : BOOL;
  /// command results
  OutCmd            : PathAccuracyModeOutCmd;    
END_VAR
VAR
  /// internal copy of command parameter 
 _parCmd             : PathAccuracyModeParCmd;
  /// command data to send
 _command            : PathAccuracyModeSendData;
  /// response data received
 _response           : PathAccuracyModeRecvData;      
END_VAR

SUPER^(AxesGroup := AxesGroup);

METHOD PROTECTED CheckFunctionSupported : BOOL
VAR_IN_OUT
  /// Robot assignment of function
  AxesGroup : AxesGroup; 
END_VAR
CheckFunctionSupported := AxesGroup.InternalData.RCSupportedFunctions.PathAccuracyMode;

IF ( NOT CheckFunctionSupported )
THEN
  // call base implementation for set error and create log entry
  SUPER^.CheckFunctionSupported(AxesGroup := AxesGroup);
END_IF
END_METHOD

METHOD PROTECTED CheckParameterChanged : BOOL
VAR_IN_OUT
  /// Robot assignment of function
  AxesGroup    : AxesGroup; 
END_VAR
// Check ParCmd Size is > 0, because MemCmp does not work correctly with size = 0
IF (SIZEOF(ParCmd) = 0) 
THEN 
  RETURN;
END_IF

// compare memory 
_parameterChanged := ( SysDepMemCmp(pData1 := ADR(ParCmd), pData2 := ADR(_parCmd), DataLen := SIZEOF(ParCmd)) <> RobotLibraryConstants.OK );

// check parameter valid ?
_parameterValid   := CheckParameterValid( AxesGroup := AxesGroup );

IF ((  _parameterChanged        )  AND 
    (  _parameterValid          )) OR
    (  _parameterUpdateInternal )  
THEN  
  // reset internal flag for send parameter update
 _parameterUpdateInternal := FALSE;
  // update internal copy of parameters 
 _parCmd := ParCmd;
  // inc parameter sequence
 _command.ParSeq := _command.ParSeq + 1;
  // update command data  
  CommandData := CreateCommandPayload(AxesGroup := AxesGroup); // ( Access via reference to rCommandFB in ACR )
  // notify active command register 
  AxesGroup.Acyclic.ActiveCommandRegister.NotifyParameterChanged := _uniqueID;
  // Reset parameter accepted flag
  ParameterAccepted := FALSE;  
END_IF
END_METHOD

METHOD INTERNAL CreateCommandPayload : RobotLibrarySendDataFB
VAR_IN_OUT
  /// Robot assignment of function
  AxesGroup : AxesGroup; 
END_VAR
// Table 6-703: Sent CMD payload (PLC to RC) of "PathAccuracyMode"
// --------------------------
// Header
// --------------------------
// Byte 00 : UINT  - Type HB     
// Byte 01 :       - Type LB    
// Byte 02 : USINT - Reserve | ExecutionMode
// Byte 03 : USINT - ParSeq  | Priority
// --------------------------
// Datablock
// --------------------------
// Byte 4  : BOOL  - Enable
// set command parameter 
_command.CmdTyp     :=  CmdType.PathAccuracyMode;
_command.ExecMode   :=  ExecMode;
_command.ParSeq     := _command.ParSeq;
_command.Priority   :=  Priority;
_command.Enable     :=  Enable;

// copy command data to header
_cmdHeader := _command;
// call base implementation to copy header to payload buffer
CreateCommandPayload := SUPER^.CreateCommandPayload(AxesGroup := AxesGroup);

// add command.Enable
CreateCommandPayload.AddBool(_command.Enable);

// Create logging
CreateCommandPayloadLog(AxesGroup := AxesGroup);
END_METHOD

METHOD INTERNAL CreateCommandPayloadLog
VAR_IN_OUT
  /// Robot assignment of function
  AxesGroup : AxesGroup; 
END_VAR
// Create log entry for Parameter start
CreateLogMessage      ( Timestamp   := AxesGroup.InternalData.SystemTime,
                        MessageType := MessageType.CMD,
                        Severity    := Severity.DEBUG,
                        MessageCode := 0,
                        MessageText := 'Create command payload with the following parameter(s) :');
  
// Create log entry for Enable
CreateLogMessagePara1 ( Timestamp   := AxesGroup.InternalData.SystemTime,
                        MessageType := MessageType.CMD,
                        Severity    := Severity.DEBUG,
                        MessageCode := 0,
                        MessageText := 'Command.Enable = {1}',
                        Para1       :=  Bool_TO_STRING(_command.Enable));
END_METHOD

METHOD FB_init : BOOL
VAR_INPUT
  /// if TRUE, the retain variables are initialized (warm start / cold start)
  bInitRetains : BOOL; 
  /// if TRUE, the instance afterwards gets moved into the copy code (online change)
  bInCopyCode  : BOOL;  
END_VAR
MyType := 'MC_PathAccuracyModeFB';

ExecMode := ExecutionMode.PARALLEL;
END_METHOD

METHOD PROTECTED OnCall
VAR_IN_OUT
  /// Robot assignment of function
  AxesGroup : AxesGroup; 
END_VAR
// call base implementation
SUPER^.OnCall(AxesGroup := AxesGroup);

CASE _stepCmd OF
  
  00:  IF ( _enable_R.Q ) 
       THEN
         // reset the rising edge
        _enable_R();       
         // reset the falling edge
        _enable_F();

         // Check function is supported and parameter are valid ?
         IF (( CheckFunctionSupported( AxesGroup := AxesGroup )) AND
             ( CheckParameterValid   ( AxesGroup := AxesGroup )))      
         THEN
           // set busy flag
           Busy := TRUE;
           // Reset command outputs
           SysDepMemSet(pDest := ADR(OutCmd), Value := 0, DataLen := SIZEOF(OutCmd));         
           // apply command parameter
          _parCmd := ParCmd;
           // init parameter sequence
          _command.ParSeq := 1;
           // create command data
           CommandData := CreateCommandPayload(AxesGroup := AxesGroup);
           // Add command to active command register
          _uniqueID := AxesGroup.Acyclic.ActiveCommandRegister.AddCmd( pCommandFB := ADR(THIS^ ));     
           // set timeout
           SetTimeout(PT := _timeoutCmd, rTimer := _timerCmd);
           // inc step counter
          _stepCmd := _stepCmd + 1; 
         END_IF   
       END_IF
     

  01:  // Wait for responce received
       IF ( _responseReceived )
       THEN
         // reset response received flag
        _responseReceived := FALSE;

         CASE  _response.State 
         OF
           CmdMessageState.BUFFERED    : CommandBuffered    := TRUE;
           CmdMessageState.ACTIVE      : ParameterAccepted  := TRUE;           
           CmdMessageState.ERROR       : Error              := TRUE;
         END_CASE
         
         // Update results
         Enabled := _response.Enabled;
                
         // Done, Aborted or Error ?
         IF (_response.State >= CmdMessageState.DONE )
         THEN
           // Reset Enabled flag
           Enabled := FALSE;
           // set timeout
           SetTimeout(PT := _timeoutCmd, rTimer := _timerCmd);
           // inc step counter
          _stepCmd := _stepCmd + 1; 
         END_IF
       END_IF

       // do not abort directly, so that the ParSeq update can be send
       IF ( _enable_R.Q ) OR ( _enable_F.Q ) 
       THEN
         // trigger parameter update to disable FB
        _parameterUpdateInternal := TRUE;
         // reset the rising edge
        _enable_R();       
         // reset the falling edge
        _enable_F();       
       END_IF

  02: IF (NOT Enable)
      THEN
        Reset();   
      END_IF

ELSE
  // invalid step
  ErrorID := RobotLibraryEvents.ERR_INVALID_STEP;
END_CASE



// Reset FB
IF (( _enable_R.Q ) OR
    ( _enable_F.Q ))
THEN
  Reset(); 
END_IF
END_METHOD

METHOD INTERNAL ParseResponsePayload : DINT
VAR_INPUT
  /// Response data
  ResponseData : RobotLibraryRecvDataFB;
  /// Timestamp
  Timestamp    : SystemTime;  
END_VAR
// Table 6-704: Received CMD payload (RC to PLC) of "PathAccuracyMode"
// --------------------------
// Header
// --------------------------
// Byte 00 : USINT - ParSeq | State     
// Byte 01 : SINT  - AlarmMessageSeverity    
// Byte 02 : UINT  - AlarmMessageCode HB
// Byte 03 :       - AlarmMessageCode LB
// --------------------------
// Datablock
// --------------------------
// Byte 04 : BOOL  - Enabled
// --------------------------
// call base implementation to parse the header from payload buffer
ResponseData.PayloadPtr := SUPER^.ParseResponsePayload(ResponseData := ResponseData, Timestamp := Timestamp);

// copy parsed header to response
_response.ParSeq               := _rspHeader.ParSeq;
_response.State                := _rspHeader.State;
_response.AlarmMessageSeverity := _rspHeader.AlarmMessageSeverity;
_response.AlarmMessageCode     := _rspHeader.AlarmMessageCode;

// Get Response.Enabled
_response.Enabled := ResponseData.GetBool();

// Create logging
ParseResponsePayloadLog(ResponseData := ResponseData, Timestamp := Timestamp);
END_METHOD

METHOD INTERNAL ParseResponsePayloadLog
VAR_INPUT
  /// Response data
  ResponseData : RobotLibraryRecvDataFB;
  /// Timestamp
  Timestamp    : SystemTime;  
END_VAR
// Create log entry for Parameter start
CreateLogMessage      ( Timestamp   := Timestamp,
                        MessageType := MessageType.CMD,
                        Severity    := Severity.DEBUG,
                        MessageCode := 0,
                        MessageText := 'Parsed the following parameter(s) from response data:');
                        
// Create log entry for Enabled
CreateLogMessagePara1 ( Timestamp   := Timestamp,
                        MessageType := MessageType.CMD,
                        Severity    := Severity.DEBUG,
                        MessageCode := 0,
                        MessageText := 'Response.Enabled = {1}',
                        Para1       :=  BOOL_TO_STRING(_response.Enabled));
END_METHOD

METHOD PROTECTED Reset : DINT
VAR_INPUT
END_VAR
Reset := SUPER^.Reset();

Busy               := FALSE;
CommandBuffered    := FALSE;
ParameterAccepted  := FALSE;
END_METHOD

END_FUNCTION_BLOCK

// Library/POUs/Additional/MC_ReadCallSubprogramCyclic/MC_ReadCallSubprogramCyclicFB
/// Reads cyclic data of called subprogram
FUNCTION_BLOCK MC_ReadCallSubprogramCyclicFB EXTENDS RobotLibraryBaseEnableFB
// ------------------------------------------------------------------------- 
//  SRCI Robot Library                                                
// ------------------------------------------------------------------------- 
//                                                                           
//  Object:      ReadCallSubprogramCyclicFB                                       
//  Author:      Thorsten Brach                                                
//  Date:        2024-06-01
//
//  Description:                                              
//   
//                                                                           
//  Copyright: 
//    (C) 2024 Thorsten Brach. All rights reserved                                                                                                                                            
//             Licensed under the LGPL-3.0 license.
//                                                                           
//  Disclaimer:                                                                           
//    This project is provided without any guarantee and can be used for   
//    private and commercial purposes. Any use is at the user’s 
//    own risk and responsibility.
//
// -------------------------------------------------------------------------
VAR_INPUT
  /// command parameter
  ParCmd  : ReadCallSubprogramCyclicParCmd;  
END_VAR

VAR_OUTPUT
  /// command outputs
  OutCmd  : ReadCallSubprogramCyclicOutCmd;  
END_VAR

SUPER^(AxesGroup := AxesGroup);

METHOD PROTECTED CheckFunctionSupported : BOOL
VAR_IN_OUT
  /// Robot assignment of function
  AxesGroup : AxesGroup; 
END_VAR
CheckFunctionSupported := AxesGroup.InternalData.RCSupportedFunctions.ReadCallSubprogramCyclic;

IF ( NOT CheckFunctionSupported )
THEN
  // call base implementation for set error and create log entry
  SUPER^.CheckFunctionSupported(AxesGroup := AxesGroup);
END_IF
END_METHOD

METHOD FB_init : BOOL
VAR_INPUT
  /// if TRUE, the retain variables are initialized (warm start / cold start)
  bInitRetains : BOOL; 
  /// if TRUE, the instance afterwards gets moved into the copy code (online change)
  bInCopyCode  : BOOL;  
END_VAR
MyType := 'MC_ReadCallSubprogramCyclicFB';
END_METHOD

METHOD PROTECTED OnCall
VAR_IN_OUT
  /// Robot assignment of function
  AxesGroup : AxesGroup; 
END_VAR
// call base implementation
SUPER^.OnCall(AxesGroup := AxesGroup);

AxesGroup.Parameter.Rob.OptionalCyclic.UseCallSubprogram := Enable;

Enabled     := AxesGroup.CyclicOptional.RobToPlc.SubProgramData.Active;
OutCmd.Data := AxesGroup.CyclicOptional.RobToPlc.SubProgramData.Data;
Busy        := (Enabled <> Enable);
END_METHOD

END_FUNCTION_BLOCK

// Library/POUs/Additional/MC_ShiftPosition/MC_ShiftPositionFB
/// Transform a defined position in space
FUNCTION_BLOCK MC_ShiftPositionFB EXTENDS RobotLibraryBaseExecuteFB
// ------------------------------------------------------------------------- 
//  SRCI Robot Library                                                
// ------------------------------------------------------------------------- 
//                                                                           
//  Object:      ShiftPositionFB                                       
//  Author:      Thorsten Brach                                                
//  Date:        2024-06-01
//
//  Description:                                              
//   
//                                                                           
//  Copyright: 
//    (C) 2024 Thorsten Brach. All rights reserved                                                                                                                                            
//             Licensed under the LGPL-3.0 license.
//                                                                           
//  Disclaimer:                                                                           
//    This project is provided without any guarantee and can be used for   
//    private and commercial purposes. Any use is at the user’s 
//    own risk and responsibility.
//
// -------------------------------------------------------------------------
VAR_INPUT
  /// Command parameter 
  ParCmd          : ShiftPositionParCmd;
END_VAR
VAR_OUTPUT
  /// Command is transferred and confirmed by the RC
  CommandBuffered : BOOL;
  /// command results
  OutCmd          : ShiftPositionOutCmd;    
END_VAR
VAR
  /// internal copy of command parameter 
 _parCmd          : ShiftPositionParCmd;
  /// command data to send
 _command         : ShiftPositionSendData;
  /// response data received
 _response        : ShiftPositionRecvData;      
END_VAR

SUPER^(AxesGroup := AxesGroup);

METHOD PROTECTED CheckFunctionSupported : BOOL
VAR_IN_OUT
  /// Robot assignment of function
  AxesGroup : AxesGroup; 
END_VAR
CheckFunctionSupported := AxesGroup.InternalData.RCSupportedFunctions.ShiftPosition;

IF ( NOT CheckFunctionSupported )
THEN
  // call base implementation for set error and create log entry
  SUPER^.CheckFunctionSupported(AxesGroup := AxesGroup);
END_IF
END_METHOD

METHOD PROTECTED CheckParameterChanged : BOOL
VAR_IN_OUT
  /// Robot assignment of function
  AxesGroup    : AxesGroup; 
END_VAR
// Check ParCmd Size is > 0, because MemCmp does not work correctly with size = 0
IF (SIZEOF(ParCmd) = 0) 
THEN 
  RETURN;
END_IF

// compare memory 
_parameterChanged := ( SysDepMemCmp(pData1 := ADR(ParCmd), pData2 := ADR(_parCmd), DataLen := SIZEOF(ParCmd)) <> RobotLibraryConstants.OK );

// check parameter valid ?
_parameterValid   := CheckParameterValid( AxesGroup := AxesGroup );

IF ((  _parameterChanged        )  AND 
    (  _parameterValid          )) OR
    (  _parameterUpdateInternal )  
THEN  
  // reset internal flag for send parameter update
 _parameterUpdateInternal := FALSE;
  // update internal copy of parameters 
 _parCmd := ParCmd;
  // inc parameter sequence
 _command.ParSeq := _command.ParSeq + 1;
  // update command data  
  CommandData := CreateCommandPayload(AxesGroup := AxesGroup); // ( Access via reference to rCommandFB in ACR )
  // notify active command register 
  AxesGroup.Acyclic.ActiveCommandRegister.NotifyParameterChanged := _uniqueID;
END_IF
END_METHOD

METHOD INTERNAL CreateCommandPayload : RobotLibrarySendDataFB
VAR_IN_OUT
  /// Robot assignment of function
  AxesGroup : AxesGroup; 
END_VAR
// Table 6-668: Sent CMD payload (PLC to RC) of "ShiftPosition"
// --------------------------
// Header
// --------------------------
// Byte 00 : UINT  - Type HB     
// Byte 01 :       - Type LB    
// Byte 02 : USINT - Reserve | ExecutionMode
// Byte 03 : USINT - ParSeq  | Priority
// --------------------------
// Datablock
// --------------------------
// Byte 04  : IEC_DATE  - TransformationParameter_1.Date
// Byte 05  :           - Reserved
// Byte 06  : IEC_TIME  - TransformationParameter_1.Time HW HB
// Byte 07  :           - TransformationParameter_1.Time HW LB
// Byte 08  :           - TransformationParameter_1.Time LW HB
// Byte 09  :           - TransformationParameter_1.Time LW LB
// Byte 10  : USINT     - TransformationParameter_1.ReferenceFrame
// Byte 11  : BYTE      - Reserved
// Byte 12  : REAL      - TransformationParameter_1.X HW HB
// Byte 13  :           - TransformationParameter_1.X HW LB
// Byte 14  :           - TransformationParameter_1.X LW HB
// Byte 15  :           - TransformationParameter_1.X LW LB
// Byte 16  : REAL      - TransformationParameter_1.Y HW HB
// Byte 17  :           - TransformationParameter_1.Y HW LB
// Byte 18  :           - TransformationParameter_1.Y LW HB
// Byte 19  :           - TransformationParameter_1.Y LW LB
// Byte 20  : REAL      - TransformationParameter_1.Z HW HB
// Byte 21  :           - TransformationParameter_1.Z HW LB
// Byte 22  :           - TransformationParameter_1.Z LW HB
// Byte 23  :           - TransformationParameter_1.Z LW LB
// Byte 24  : REAL      - TransformationParameter_1.RX HW HB
// Byte 25  :           - TransformationParameter_1.RX HW LB
// Byte 26  :           - TransformationParameter_1.RX LW HB
// Byte 27  :           - TransformationParameter_1.RX LW LB
// Byte 28  : REAL      - TransformationParameter_1.RY HW HB
// Byte 29  :           - TransformationParameter_1.RY HW LB
// Byte 30  :           - TransformationParameter_1.RY LW HB
// Byte 31  :           - TransformationParameter_1.RY LW LB
// Byte 32  : REAL      - TransformationParameter_1.RZ HW HB
// Byte 33  :           - TransformationParameter_1.RZ HW LB
// Byte 34  :           - TransformationParameter_1.RZ LW HB
// Byte 35  :           - TransformationParameter_1.RZ LW LB
// Byte 36  : USINT     - TransformationParameter_2
// Byte 37  : REAL      - RotationAngle HW HB
// Byte 38  :           - RotationAngle HW LB
// Byte 39  :           - RotationAngle LW HB
// Byte 40  :           - RotationAngle LW LB
// Byte 41  : SINT      - Mode
// Byte 42  : USINT     - FrameNo
// Byte 43  : USINT     - TargetFrameNo
// Byte 44  : REAL      - Position.X HW HB
// Byte 45  :           - Position.X HW LB
// Byte 46  :           - Position.X LW HB
// Byte 47  :           - Position.X LW LB
// Byte 48  : REAL      - Position.Y HW HB
// Byte 49  :           - Position.Y HW LB
// Byte 50  :           - Position.Y LW HB
// Byte 51  :           - Position.Y LW LB
// Byte 52  : REAL      - Position.Z HW HB
// Byte 53  :           - Position.Z HW LB
// Byte 54  :           - Position.Z LW HB
// Byte 55  :           - Position.Z LW LB
// Byte 56  : REAL      - Position.RX HW HB
// Byte 57  :           - Position.RX HW LB
// Byte 58  :           - Position.RX LW HB
// Byte 59  :           - Position.RX LW LB
// Byte 60  : REAL      - Position.RY HW HB
// Byte 61  :           - Position.RY HW LB
// Byte 62  :           - Position.RY LW HB
// Byte 63  :           - Position.RY LW LB
// Byte 64  : REAL      - Position.RZ HW HB
// Byte 65  :           - Position.RZ HW LB
// Byte 66  :           - Position.RZ LW HB
// Byte 67  :           - Position.RZ LW LB
// Byte 68  : ArmConfig - Position.Config
// Byte 69  :           -          Reserve
// Byte 70 : TurnNumber - Position.TurnNumber.J1 + J2  HW HB
// Byte 71 :            - Position.TurnNumber.J3 + J4  HW LB
// Byte 72 :            - Position.TurnNumber.J5 + J6  LW LB
// Byte 73 :            - Position.TurnNumber.E1       LW LB
// Byte 74  : REAL      - Position.E1 HW HB
// Byte 75  :           - Position.E1 HW LB
// Byte 76  :           - Position.E1 LW HB
// Byte 77  :           - Position.E1 LW LB
// Byte 78  : REAL      - Position.E2 HW HB
// Byte 79  :           - Position.E2 HW LB
// Byte 80  :           - Position.E2 LW HB
// Byte 81  :           - Position.E2 LW LB
// Byte 82  : REAL      - Position.E3 HW HB
// Byte 83  :           - Position.E3 HW LB
// Byte 84  :           - Position.E3 LW HB
// Byte 85  :           - Position.E3 LW LB
// Byte 86  : REAL      - Position.E4 HW HB
// Byte 87  :           - Position.E4 HW LB
// Byte 88  :           - Position.E4 LW HB
// Byte 89  :           - Position.E4 LW LB
// Byte 90  : REAL      - Position.E5 HW HB
// Byte 91  :           - Position.E5 HW LB
// Byte 92  :           - Position.E5 LW HB
// Byte 93  :           - Position.E5 LW LB
// Byte 94  : REAL      - Position.E6 HW HB
// Byte 95  :           - Position.E6 HW LB
// Byte 96  :           - Position.E6 LW HB
// Byte 97  :           - Position.E6 LW LB
// set command parameter 
_command.CmdTyp                    :=  CmdType.ShiftPosition;
_command.ExecMode                  :=  ExecMode;
_command.ParSeq                    := _command.ParSeq;
_command.Priority                  :=  Priority;
_command.TransformationParameter_1 := _parCmd.TransformationParameter_1;
_command.TransformationParameter_2 := _parCmd.TransformationParameter_2;
_command.RotationAngle             := _parCmd.RotationAngle;
_command.Mode                      := _parCmd.Mode;
_command.FrameNo                   := _parCmd.FrameNo;
_command.TargetFrameNo             := _parCmd.TargetFrameNo;
_command.Position                  := _parCmd.Position;

// copy command data to header
_cmdHeader := _command;
// call base implementation to copy header to payload buffer
CreateCommandPayload := SUPER^.CreateCommandPayload(AxesGroup := AxesGroup);

// add command.TransformationParameter_1.Timestamp.IEC_DATE
CreateCommandPayload.AddIecDate(_command.TransformationParameter_1.Timestamp.IEC_DATE);
// add command.TransformationParameter_1.Timestamp.IEC_TIME
CreateCommandPayload.AddIecTime(_command.TransformationParameter_1.Timestamp.IEC_TIME);
// add command.TransformationParameter_1.ReferenceFrame
CreateCommandPayload.AddUsint(_command.TransformationParameter_1.ReferenceFrame);
// add command.Reserve
CreateCommandPayload.AddByte(0);
// add command.TransformationParameter_1.X
CreateCommandPayload.AddReal(_command.TransformationParameter_1.X);
// add command.TransformationParameter_1.Y
CreateCommandPayload.AddReal(_command.TransformationParameter_1.Y);
// add command.TransformationParameter_1.Z
CreateCommandPayload.AddReal(_command.TransformationParameter_1.Z);
// add command.TransformationParameter_1.Rx
CreateCommandPayload.AddReal(_command.TransformationParameter_1.Rx);
// add command.TransformationParameter_1.Ry
CreateCommandPayload.AddReal(_command.TransformationParameter_1.Ry);
// add command.TransformationParameter_1.Rz
CreateCommandPayload.AddReal(_command.TransformationParameter_1.Rz);
// add command.TransformationParameter_2
CreateCommandPayload.AddUsint(_command.TransformationParameter_2);
// add command.RotationAngle
CreateCommandPayload.AddReal(_command.RotationAngle);
// add command.Mode
CreateCommandPayload.AddSint(_command.Mode);
// add command.FrameNo
CreateCommandPayload.AddUsint(_command.FrameNo);
// add command.TargetFrameNo
CreateCommandPayload.AddUsint(_command.TargetFrameNo);
// add command.Position.X
CreateCommandPayload.AddReal(_command.Position.X);
// add command.Position.Y
CreateCommandPayload.AddReal(_command.Position.Y);
// add command.Position.Z
CreateCommandPayload.AddReal(_command.Position.Z);
// add command.Position.Rx
CreateCommandPayload.AddReal(_command.Position.Rx);
// add command.Position.Ry
CreateCommandPayload.AddReal(_command.Position.Ry);
// add command.Position.Rz
CreateCommandPayload.AddReal(_command.Position.Rz);
// add command.Position.Config
CreateCommandPayload.AddArmConfig(_command.Position.Config);
// add command.Position.Config
CreateCommandPayload.AddTurnNumber(_command.Position.TurnNumber);
// add command.Position.E1
CreateCommandPayload.AddReal(_command.Position.E1);
// add command.Position.E2
CreateCommandPayload.AddReal(_command.Position.E2);
// add command.Position.E3
CreateCommandPayload.AddReal(_command.Position.E3);
// add command.Position.E4
CreateCommandPayload.AddReal(_command.Position.E4);
// add command.Position.E5
CreateCommandPayload.AddReal(_command.Position.E5);
// add command.Position.E6
CreateCommandPayload.AddReal(_command.Position.E6);

// Create logging
CreateCommandPayloadLog(AxesGroup := AxesGroup);
END_METHOD

METHOD INTERNAL CreateCommandPayloadLog
VAR_IN_OUT
  /// Robot assignment of function
  AxesGroup : AxesGroup; 
END_VAR
// Create log entry for Parameter start
CreateLogMessage      ( Timestamp   := AxesGroup.InternalData.SystemTime,
                        MessageType := MessageType.CMD,
                        Severity    := Severity.DEBUG,
                        MessageCode := 0,
                        MessageText := 'Create command payload with the following parameter(s) :');
  
// Create log entry for TransformationParameter_1.Timestamp.IEC_DATE
CreateLogMessagePara1 ( Timestamp   := AxesGroup.InternalData.SystemTime,
                        MessageType := MessageType.CMD,
                        Severity    := Severity.DEBUG,
                        MessageCode := 0,
                        MessageText := 'Command.TransformationParameter_1.Timestamp.IEC_DATE = {1}',
                        Para1       :=  IEC_DATE_TO_STRING(_command.TransformationParameter_1.Timestamp.IEC_DATE));
                       
// Create log entry for TransformationParameter_1.Timestamp.IEC_TIME
CreateLogMessagePara1 ( Timestamp   := AxesGroup.InternalData.SystemTime,
                        MessageType := MessageType.CMD,
                        Severity    := Severity.DEBUG,
                        MessageCode := 0,
                        MessageText := 'Command.TransformationParameter_1.Timestamp.IEC_TIME = {1}',
                        Para1       :=  IEC_TIME_TO_STRING(_command.TransformationParameter_1.Timestamp.IEC_TIME));

// Create log entry for TransformationParameter_1.ReferenceFrame
CreateLogMessagePara1 ( Timestamp   := AxesGroup.InternalData.SystemTime,
                        MessageType := MessageType.CMD,
                        Severity    := Severity.DEBUG,
                        MessageCode := 0,
                        MessageText := 'Command.TransformationParameter_1.ReferenceFrame = {1}',
                        Para1       :=  USINT_TO_STRING(_command.TransformationParameter_1.ReferenceFrame));

// Create log entry for Reserve
CreateLogMessagePara1 ( Timestamp   := AxesGroup.InternalData.SystemTime,
                        MessageType := MessageType.CMD,
                        Severity    := Severity.DEBUG,
                        MessageCode := 0,
                        MessageText := 'Command.Reserve = {1}',
                        Para1       :=  USINT_TO_STRING(0));

// Create log entry for TransformationParameter_1.X
CreateLogMessagePara1 ( Timestamp   := AxesGroup.InternalData.SystemTime,
                        MessageType := MessageType.CMD,
                        Severity    := Severity.DEBUG,
                        MessageCode := 0,
                        MessageText := 'Command.TransformationParameter_1.X = {1}',
                        Para1       :=  REAL_TO_STRING(_command.TransformationParameter_1.X));

// Create log entry for TransformationParameter_1.Y
CreateLogMessagePara1 ( Timestamp   := AxesGroup.InternalData.SystemTime,
                        MessageType := MessageType.CMD,
                        Severity    := Severity.DEBUG,
                        MessageCode := 0,
                        MessageText := 'Command.TransformationParameter_1.Y = {1}',
                        Para1       :=  REAL_TO_STRING(_command.TransformationParameter_1.Y));
                       
// Create log entry for TransformationParameter_1.Z
CreateLogMessagePara1 ( Timestamp   := AxesGroup.InternalData.SystemTime,
                        MessageType := MessageType.CMD,
                        Severity    := Severity.DEBUG,
                        MessageCode := 0,
                        MessageText := 'Command.TransformationParameter_1.Z = {1}',
                        Para1       :=  REAL_TO_STRING(_command.TransformationParameter_1.Z));

// Create log entry for TransformationParameter_1.Rx
CreateLogMessagePara1 ( Timestamp   := AxesGroup.InternalData.SystemTime,
                        MessageType := MessageType.CMD,
                        Severity    := Severity.DEBUG,
                        MessageCode := 0,
                        MessageText := 'Command.TransformationParameter_1.Rx = {1}',
                        Para1       :=  REAL_TO_STRING(_command.TransformationParameter_1.Rx));

// Create log entry for TransformationParameter_1.Ry
CreateLogMessagePara1 ( Timestamp   := AxesGroup.InternalData.SystemTime,
                        MessageType := MessageType.CMD,
                        Severity    := Severity.DEBUG,
                        MessageCode := 0,
                        MessageText := 'Command.TransformationParameter_1.Ry = {1}',
                        Para1       :=  REAL_TO_STRING(_command.TransformationParameter_1.Ry));

// Create log entry for TransformationParameter_1.Rz
CreateLogMessagePara1 ( Timestamp   := AxesGroup.InternalData.SystemTime,
                        MessageType := MessageType.CMD,
                        Severity    := Severity.DEBUG,
                        MessageCode := 0,
                        MessageText := 'Command.TransformationParameter_1.Rz = {1}',
                        Para1       :=  REAL_TO_STRING(_command.TransformationParameter_1.Rz));

// Create log entry for TransformationParameter_2
CreateLogMessagePara1 ( Timestamp   := AxesGroup.InternalData.SystemTime,
                        MessageType := MessageType.CMD,
                        Severity    := Severity.DEBUG,
                        MessageCode := 0,
                        MessageText := 'Command.TransformationParameter_2 = {1}',
                        Para1       :=  USINT_TO_STRING(_command.TransformationParameter_2));

// Create log entry for RotationAngle
CreateLogMessagePara1 ( Timestamp   := AxesGroup.InternalData.SystemTime,
                        MessageType := MessageType.CMD,
                        Severity    := Severity.DEBUG,
                        MessageCode := 0,
                        MessageText := 'Command.RotationAngle = {1}',
                        Para1       :=  REAL_TO_STRING(_command.RotationAngle));

// Create log entry for Mode
CreateLogMessagePara1 ( Timestamp   := AxesGroup.InternalData.SystemTime,
                        MessageType := MessageType.CMD,
                        Severity    := Severity.DEBUG,
                        MessageCode := 0,
                        MessageText := 'Command.Mode = {1}',
                        Para1       :=  TRANSFORM_MODE_TO_STRING(_command.Mode));

// Create log entry for FrameNo
CreateLogMessagePara1 ( Timestamp   := AxesGroup.InternalData.SystemTime,
                        MessageType := MessageType.CMD,
                        Severity    := Severity.DEBUG,
                        MessageCode := 0,
                        MessageText := 'Command.FrameNo = {1}',
                        Para1       :=  USINT_TO_STRING(_command.FrameNo));

// Create log entry for TargetFrameNo
CreateLogMessagePara1 ( Timestamp   := AxesGroup.InternalData.SystemTime,
                        MessageType := MessageType.CMD,
                        Severity    := Severity.DEBUG,
                        MessageCode := 0,
                        MessageText := 'Command.TargetFrameNo = {1}',
                        Para1       :=  USINT_TO_STRING(_command.TargetFrameNo));
                        
// Create log entry for Position.X
CreateLogMessagePara1 ( Timestamp   := AxesGroup.InternalData.SystemTime,
                        MessageType := MessageType.CMD,
                        Severity    := Severity.DEBUG,
                        MessageCode := 0,
                        MessageText := 'Command.Position.X = {1}',
                        Para1       :=  REAL_TO_STRING(_command.Position.X));

// Create log entry for Position.Y
CreateLogMessagePara1 ( Timestamp   := AxesGroup.InternalData.SystemTime,
                        MessageType := MessageType.CMD,
                        Severity    := Severity.DEBUG,
                        MessageCode := 0,
                        MessageText := 'Command.Position.Y = {1}',
                        Para1       :=  REAL_TO_STRING(_command.Position.Y));

// Create log entry for Position.Z
CreateLogMessagePara1 ( Timestamp   := AxesGroup.InternalData.SystemTime,
                        MessageType := MessageType.CMD,
                        Severity    := Severity.DEBUG,
                        MessageCode := 0,
                        MessageText := 'Command.Position.Z = {1}',
                        Para1       :=  REAL_TO_STRING(_command.Position.Z));

// Create log entry for Position.Rx
CreateLogMessagePara1 ( Timestamp   := AxesGroup.InternalData.SystemTime,
                        MessageType := MessageType.CMD,
                        Severity    := Severity.DEBUG,
                        MessageCode := 0,
                        MessageText := 'Command.Position.Rx = {1}',
                        Para1       :=  REAL_TO_STRING(_command.Position.Rx));

// Create log entry for Position.Ry
CreateLogMessagePara1 ( Timestamp   := AxesGroup.InternalData.SystemTime,
                        MessageType := MessageType.CMD,
                        Severity    := Severity.DEBUG,
                        MessageCode := 0,
                        MessageText := 'Command.Position.Ry = {1}',
                        Para1       :=  REAL_TO_STRING(_command.Position.Ry));

// Create log entry for Position.Rz
CreateLogMessagePara1 ( Timestamp   := AxesGroup.InternalData.SystemTime,
                        MessageType := MessageType.CMD,
                        Severity    := Severity.DEBUG,
                        MessageCode := 0,
                        MessageText := 'Command.Position.Rz = {1}',
                        Para1       :=  REAL_TO_STRING(_command.Position.Rz));
                        
// Create log entry for Position.Config
CreateLogMessagePara1 ( Timestamp   := AxesGroup.InternalData.SystemTime,
                        MessageType := MessageType.CMD,
                        Severity    := Severity.DEBUG,
                        MessageCode := 0,
                        MessageText := 'Command.Config = {1}',
                        Para1       :=  ARM_CONFIG_TO_STRING(_command.Position.Config));

// Create log entry for Position.TurnNumber[0]
CreateLogMessagePara1 ( Timestamp   := AxesGroup.InternalData.SystemTime,
                        MessageType := MessageType.CMD,
                        Severity    := Severity.DEBUG,
                        MessageCode := 0,
                        MessageText := 'Command.Position.TurnNumber[0] = {1}',
                        Para1       :=  BYTE_TO_STRING(CombineHalfSints(HalfSintHi := _command.Position.TurnNumber.J2Turns, 
                                                                        HalfSintLo := _command.Position.TurnNumber.J1Turns)));

// Create log entry for Position.TurnNumber[1]
CreateLogMessagePara1 ( Timestamp   := AxesGroup.InternalData.SystemTime,
                        MessageType := MessageType.CMD,
                        Severity    := Severity.DEBUG,
                        MessageCode := 0,
                        MessageText := 'Command.Position.TurnNumber[1] = {1}',
                        Para1       :=  BYTE_TO_STRING(CombineHalfSints(HalfSintHi := _command.Position.TurnNumber.J4Turns, 
                                                                        HalfSintLo := _command.Position.TurnNumber.J3Turns)));

// Create log entry for Position.TurnNumber[2]
CreateLogMessagePara1 ( Timestamp   := AxesGroup.InternalData.SystemTime,
                        MessageType := MessageType.CMD,
                        Severity    := Severity.DEBUG,
                        MessageCode := 0,
                        MessageText := 'Command.Position.TurnNumber[2] = {1}',
                        Para1       :=  BYTE_TO_STRING(CombineHalfSints(HalfSintHi := _command.Position.TurnNumber.J6Turns,
                                                                        HalfSintLo := _command.Position.TurnNumber.J5Turns)));

// Create log entry for Position.TurnNumber[3]
CreateLogMessagePara1 ( Timestamp   := AxesGroup.InternalData.SystemTime,
                        MessageType := MessageType.CMD,
                        Severity    := Severity.DEBUG,
                        MessageCode := 0,
                        MessageText := 'Command.Position.TurnNumber[3] = {1}',
                        Para1       :=  SINT_TO_STRING(_command.Position.TurnNumber.E1Turns));

// Create log entry for Position.E1
CreateLogMessagePara1 ( Timestamp   := AxesGroup.InternalData.SystemTime,
                        MessageType := MessageType.CMD,
                        Severity    := Severity.DEBUG,
                        MessageCode := 0,
                        MessageText := 'Command.Position.E1 = {1}',
                        Para1       :=  REAL_TO_STRING(_command.Position.E1));

// Create log entry for Position.E2
CreateLogMessagePara1 ( Timestamp   := AxesGroup.InternalData.SystemTime,
                        MessageType := MessageType.CMD,
                        Severity    := Severity.DEBUG,
                        MessageCode := 0,
                        MessageText := 'Command.Position.E2 = {1}',
                        Para1       :=  REAL_TO_STRING(_command.Position.E2));

// Create log entry for Position.E3
CreateLogMessagePara1 ( Timestamp   := AxesGroup.InternalData.SystemTime,
                        MessageType := MessageType.CMD,
                        Severity    := Severity.DEBUG,
                        MessageCode := 0,
                        MessageText := 'Command.Position.E3 = {1}',
                        Para1       :=  REAL_TO_STRING(_command.Position.E3));

// Create log entry for Position.E4
CreateLogMessagePara1 ( Timestamp   := AxesGroup.InternalData.SystemTime,
                        MessageType := MessageType.CMD,
                        Severity    := Severity.DEBUG,
                        MessageCode := 0,
                        MessageText := 'Command.Position.E4 = {1}',
                        Para1       :=  REAL_TO_STRING(_command.Position.E4));
                        
// Create log entry for Position.E5
CreateLogMessagePara1 ( Timestamp   := AxesGroup.InternalData.SystemTime,
                        MessageType := MessageType.CMD,
                        Severity    := Severity.DEBUG,
                        MessageCode := 0,
                        MessageText := 'Command.Position.E5 = {1}',
                        Para1       :=  REAL_TO_STRING(_command.Position.E5));

// Create log entry for Position.E6
CreateLogMessagePara1 ( Timestamp   := AxesGroup.InternalData.SystemTime,
                        MessageType := MessageType.CMD,
                        Severity    := Severity.DEBUG,
                        MessageCode := 0,
                        MessageText := 'Command.Position.E6 = {1}',
                        Para1       :=  REAL_TO_STRING(_command.Position.E6));
END_METHOD

METHOD FB_init : BOOL
VAR_INPUT
  /// if TRUE, the retain variables are initialized (warm start / cold start)
  bInitRetains : BOOL; 
  /// if TRUE, the instance afterwards gets moved into the copy code (online change)
  bInCopyCode  : BOOL;  
END_VAR
MyType := 'MC_ShiftPositionFB';

ExecMode := ExecutionMode.PARALLEL;
END_METHOD

METHOD PROTECTED OnCall
VAR_IN_OUT
  /// Robot assignment of function
  AxesGroup : AxesGroup; 
END_VAR
// call base implementation
SUPER^.OnCall(AxesGroup := AxesGroup);

CASE _stepCmd OF
  
